// POUs/LinMot Config Function Blocks/LMcf_GetModUPIDList
FUNCTION_BLOCK LMcf_GetModUPIDList
VAR_INPUT
	Execute			:BOOL; 	(*Execute command*)
	adrFirstEntry	:POINTER TO tstLM_CfgUPIDListEntry; (*Points to the first entry of an array of UPIDListEntries (UPIDs and the according UPID values)*)
	NrOfEntries		:UINT; 	(*Number of parameters to be read. ATTENTION: Make sure the array at FirstEntry is big enough!!!!!*)
END_VAR
VAR_IN_OUT
	Axis			:tstLM_Axis; (*Axis reference*)
END_VAR
VAR_OUTPUT
	Done			:BOOL;	(*Command has been executed*)
	Busy			:BOOL;	(*Command running / FB Busy*)
	Error			:BOOL;	(*Error occured in FB*)
	ErrorID			:UINT;	(*Error ID:
							01h: Timeout (No Response from the drive)
							02h: ConfigChannel already busy
							05h: NrOfEntries must be greater than 0 (zero)! (UPID List)
							06h: Address of UPIDListEntry array is zero! Check adrFirstEntry input! (UPID List)
 							C0h: UPID Error 
 							C1h: Parameter Type Error
 							C2h: Range Error
 							C3h: Address Usage Error
 							C5h: Error: Command 21h
 							D0h: Odd Address
 							D1h: Size Error (Curve Service)
 							D4h: Curve already defined / Curve not present (Curve Service)
							>D4h: Contact LinMot Support
							*)
END_VAR
VAR
	uiState			:UINT;	(*internal -> *)
	i				:UINT;	(*internal -> *)
	pEntry			:POINTER TO tstLM_CfgUPIDListEntry; (*internal -> *)
	fStartTrig		:LM_R_TRIG;	(*internal -> *)
	fTimer			:TON;	(*internal -> *)
	tiT1			:TIME:=T#5000ms; (*internal -> timeout*)
END_VAR
(*Version history:
Date         	 | Version    	| Created under     		| Author          		| Remark 
------------------------------------------------------------------------------------------------------------------------------- 
2011-jul-12   	 | 1.0.0      	| V2.11.0 (Build 1016)		| fj  					| initial release 
*)

(*Check on errors*)
IF ((SHR(Axis.DrvToPlc.CfgStatusWord,8) = 16#C0)
	OR (SHR(Axis.DrvToPlc.CfgStatusWord,8) = 16#C1)
	OR (SHR(Axis.DrvToPlc.CfgStatusWord,8) = 16#C2)
	OR (SHR(Axis.DrvToPlc.CfgStatusWord,8) = 16#C3)
	OR (SHR(Axis.DrvToPlc.CfgStatusWord,8) = 16#C5)
	OR (SHR(Axis.DrvToPlc.CfgStatusWord,8) = 16#D0)
	OR (SHR(Axis.DrvToPlc.CfgStatusWord,8) = 16#D1)
	OR (SHR(Axis.DrvToPlc.CfgStatusWord,8) = 16#D4)
	OR (SHR(Axis.DrvToPlc.CfgStatusWord,8) > 16#D4))
	AND uiState > 1
	AND Busy THEN
	ErrorID := SHR(Axis.DrvToPlc.CfgStatusWord, 8);
	uiState := 90;
END_IF

(*Check start trigger*)
fStartTrig(CLK:=Execute);
IF fStartTrig.Q AND NOT Busy THEN
	IF Axis.ConfigChannelBusy THEN (*Check ConfigChannel busy*)
		ErrorID := 16#02; (*Error: ConfigChannel already busy*)
		uiState := 90; (*Error*)
	ELSIF NrOfEntries <= 0 THEN
		ErrorID := 16#05; (*Error: NrOfEntries must be greater than 0 (zero)! (UPID List)*)
		uiState := 90; (*Error*)
	ELSIF adrFirstEntry = 0 THEN
		ErrorID := 16#06; (*Address of UPIDListEntry array is zero! Check adrFirstEntry input! (UPID List)*)
		uiState := 90; (*Error*)
	ELSE
		Axis.ConfigChannelBusy := TRUE;
		Busy := TRUE;
		uiState := 1;
	END_IF
END_IF

(*State machine*)
CASE uiState OF
	(*Idle state*)
	0: 	;

(*=============================================================================
*  Get Modified UPID List
===============================================================================*)

	(*Prepare Config Module*)
	1: 	Axis.PlcToDrv.CfgControlWord := 16#000F;
		Axis.PlcToDrv.CfgIndexOut := 16#0000;
		Axis.PlcToDrv.CfgValueOut := 16#00000000;
		fTimer(IN:=TRUE,PT:=tiT1);

		pEntry := adrFirstEntry; (*Copy pointer*)
		i := 0; (*Reset i*)

		IF fTimer.Q THEN
			fTimer(IN:=FALSE);
			ErrorID := 16#01; (*fTimer error: No response from drive*)
			uiState := 90;
		END_IF

		IF Axis.DrvToPlc.CfgStatusWord = 16#000F THEN
			fTimer(IN:=FALSE);
			uiState := 2;
		END_IF

	 (*Start Getting Modified UPID List*)
	2:	Axis.PlcToDrv.CfgControlWord := 16#2201;
		fTimer(IN:=TRUE,PT:=tiT1);

		IF fTimer.Q THEN
			fTimer(IN:=FALSE);
			ErrorID := 16#01; (*fTimer error: No response from drive*)
			uiState := 90;
		END_IF

		IF Axis.DrvToPlc.CfgStatusWord = 16#0001 THEN
			fTimer(IN:=FALSE);
			uiState := 3;
		END_IF

	 (*Get Next Modified UPID List Item*)
	3:	Axis.PlcToDrv.CfgControlWord := 16#2302;
		fTimer(IN:=TRUE,PT:=tiT1);

		IF fTimer.Q THEN
			fTimer(IN:=FALSE);
			ErrorID := 16#01; (*fTimer error: No response from drive*)
			uiState := 90;
		END_IF

		IF Axis.DrvToPlc.CfgStatusWord = 16#C602 THEN (*End of UPID list reached*)
			fTimer(IN:=FALSE);
			pEntry^.UPID := Axis.DrvToPlc.CfgIndexIn; (*Read last UPID*)
			pEntry^.UPIDValue := Axis.DrvToPlc.CfgValueIn;
			i := i+1;
			uiState := 100;
		ELSIF Axis.DrvToPlc.CfgStatusWord = 16#0002 THEN (*UPID found*)
			fTimer(IN:=FALSE);
			pEntry^.UPID := Axis.DrvToPlc.CfgIndexIn;
			pEntry^.UPIDValue := Axis.DrvToPlc.CfgValueIn;
			pEntry := pEntry + (SIZEOF(adrFirstEntry^)); (*Increment pointer*)	
			i := i+1;
			IF i >= NrOfEntries THEN
				uiState := 100; (*Stop reading*)
			ELSE
				uiState := 4; (*Read next UPID*)
			END_IF
		END_IF

	(*Get Next Modified UPID List Item*)
	4:	Axis.PlcToDrv.CfgControlWord := 16#2303;
		fTimer(IN:=TRUE,PT:=tiT1);

		IF fTimer.Q THEN
			fTimer(IN:=FALSE);
			ErrorID := 16#01; (*fTimer error: No response from drive*)
			uiState := 90;
		END_IF

		IF Axis.DrvToPlc.CfgStatusWord = 16#C603 THEN (*End of UPID list reached*)
			fTimer(IN:=FALSE);
			pEntry^.UPID := Axis.DrvToPlc.CfgIndexIn; (*Read last UPID*)
			pEntry^.UPIDValue := Axis.DrvToPlc.CfgValueIn;
			i := i+1;
			uiState := 100;
		ELSIF Axis.DrvToPlc.CfgStatusWord = 16#0003 THEN (*UPID found*)
			fTimer(IN:=FALSE);
			pEntry^.UPID := Axis.DrvToPlc.CfgIndexIn;
			pEntry^.UPIDValue := Axis.DrvToPlc.CfgValueIn;
			pEntry := pEntry + (SIZEOF(adrFirstEntry^)); (*Increment pointer*)	
			i := i+1;
			IF i >= NrOfEntries THEN
				uiState := 100; (*Stop reading*)
			ELSE
				uiState := 3; (*Read next UPID*)
			END_IF
		END_IF

(*=============================================================================
*  Error State
===============================================================================*)    

	(*Error state I*)
	90:	IF Busy THEN
			Axis.ConfigChannelBusy := FALSE; (*Only reset ConfigChannelBusy if function block is Busy*)
			Axis.PlcToDrv.CfgControlWord := 16#0000; (*Reset Config Control*)
		END_IF

		Error := TRUE;
		Busy := FALSE;
		Done := FALSE;
		fTimer(IN:=FALSE);
		(*i := 0;*)

		uiState := 91;

	(*Error State II*)
	91:	IF NOT Execute THEN
			Error := FALSE;
			ErrorID := 0;
			uiState := 0;
		END_IF

(*=============================================================================
*  Command Done
===============================================================================*)    

	(*Command succesfully executed*)
	100:Done := TRUE;
		Busy := FALSE;
		fTimer(IN:=FALSE);
		(*i := 0;*)

		Axis.ConfigChannelBusy := FALSE;
		Axis.PlcToDrv.CfgControlWord := 16#0000; (*Reset Config Control*)

		uiState := 101;

	(*Wait Not Execute*)
	101:IF NOT Execute THEN
			Done := FALSE;
			uiState := 0;
		END_IF

END_CASE

END_FUNCTION_BLOCK

// POUs/LinMot Config Function Blocks/LMcf_ParaAccess
FUNCTION_BLOCK LMcf_ParaAccess
VAR_INPUT
	Execute			:BOOL;	(*Execute command*)
	Mode			:UINT;	(*Mode 0: Read ROM Value of Parameter by UPID [Inputs used: UPIDIn]
 							Mode 1: Read RAM Value of Parameter by UPID [Inputs used: UPIDIn]
 							Mode 2: Write ROM Value of Parameter by UPID [Inputs used: UPIDIn, ValueIn]
 							Mode 3: Write RAM Value of Parameter by UPID [Inputs used: UPIDIn, ValueIn]
 							Mode 4: Write RAM and ROM Value of Parameter by UPID [Inputs used: UPIDIn, ValueIn]
 							Mode 5: Get minimal Value of Parameter by UPID [Inputs used: UPIDIn]
 							Mode 6: Get maximal Value of Parameter by UPID [Inputs used: UPIDIn]
 							Mode 7: Get default Value of Parameter by UPID [Inputs used: UPIDIn]
							*)
	UPIDIn			:UINT;	(*UPID to access*)
	ValueIn			:DINT;	(*UPID value to be written*)
END_VAR
VAR_IN_OUT
	Axis			:tstLM_Axis; (*Axis reference*)
END_VAR
VAR_OUTPUT
	Done			:BOOL;	(*Command has been executed*)
	Busy			:BOOL;	(*Command running / FB Busy*)
	ValueOut		:DINT;	(*UPID value from drive*)
	Error			:BOOL;	(*Error occured in FB*)
	ErrorID			:UINT;	(*Error ID:
							01h: Timeout (No Response from the drive)
							02h: ConfigChannel already busy
							03h: Invalid Mode selected
 							C0h: UPID Error 
 							C1h: Parameter Type Error
 							C2h: Range Error
 							C3h: Address Usage Error
 							C5h: Error: Command 21h
 							D0h: Odd Address
 							D1h: Size Error (Curve Service)
 							D4h: Curve already defined / Curve not present (Curve Service)
							>D4h: Contact LinMot Support
							*)
END_VAR
VAR
	uiState			:UINT;	(*internal -> *)
	uiStartState	:UINT;	(*internal -> *)
	fStartTrig		:LM_R_TRIG;	(*internal -> *)
	fTimer			:TON;	(*internal -> *)
	tiT1			:TIME:=T#5000MS; (*internal -> timeout*)
END_VAR
(*Version history:
Date         	 | Version    	| Created under     		| Author          		| Remark 
------------------------------------------------------------------------------------------------------------------------------- 
2011-jul-12   	 | 1.0.0      		| V2.11.0 (Build 1016)	| fj  				| initial release 
*)

(*Check on errors*)
IF ((SHR(Axis.DrvToPlc.CfgStatusWord,8) = 16#C0)
	OR (SHR(Axis.DrvToPlc.CfgStatusWord,8) = 16#C1)
	OR (SHR(Axis.DrvToPlc.CfgStatusWord,8) = 16#C2)
	OR (SHR(Axis.DrvToPlc.CfgStatusWord,8) = 16#C3)
	OR (SHR(Axis.DrvToPlc.CfgStatusWord,8) = 16#C5)
	OR (SHR(Axis.DrvToPlc.CfgStatusWord,8) = 16#D0)
	OR (SHR(Axis.DrvToPlc.CfgStatusWord,8) = 16#D1)
	OR (SHR(Axis.DrvToPlc.CfgStatusWord,8) = 16#D4)
	OR (SHR(Axis.DrvToPlc.CfgStatusWord,8) > 16#D4))
	AND uiState > 1
	AND Busy THEN
	ErrorID := SHR(Axis.DrvToPlc.CfgStatusWord, 8);
	uiState := 90;
END_IF

(*Mode selection and edge detection*)
fStartTrig(CLK:=Execute);
IF fStartTrig.Q AND NOT Busy THEN
	CASE Mode OF
		(*Read ROM Value of Parameter by UPID*)
		0: 	uiStartState := 2;
			uiState := 1;
		(*Read RAM Value of Parameter by UPID*)
		1: 	uiStartState := 10;
			uiState := 1;
		(*Write ROM Value of Parameter by UPID*)
		2: 	uiStartState := 20;
			uiState := 1;
		(*Write RAM Value of Parameter by UPID*)
		3: 	uiStartState := 30;
			uiState := 1;
		(*Write RAM and ROM Value of Parameter by UPID*)
		4: 	uiStartState := 40;
			uiState := 1;
		(*Get minimal Value of Parameter by UPID*)
		5: 	uiStartState := 50;
			uiState := 1;
		(*Get maximal Value of Parameter by UPID*)
		6: 	uiStartState := 60;
			uiState := 1;
		(*Get default Value of Parameter by UPID*)
		7: 	uiStartState := 70;
			uiState := 1;
		ELSE ;
	END_CASE

	IF Axis.ConfigChannelBusy THEN (*Check ConfigChannel busy*)
		ErrorID := 16#02; (*Error: ConfigChannel already busy*)
		uiState := 90; (*Error*)
	ELSIF Mode > 7 THEN
		ErrorID := 16#03; (*Error: Invalid Mode selected*)
		uiState := 90; (*Error*)
	ELSE
		Axis.ConfigChannelBusy := TRUE;
		Busy := TRUE;
	END_IF
END_IF

(*State machine*)
CASE uiState OF
	(*Idle state*)
	0: 	;

	(*Prepare Config Module*)
	1: 	Axis.PlcToDrv.CfgControlWord := 16#000F;
		Axis.PlcToDrv.CfgIndexOut := 16#0000;
		Axis.PlcToDrv.CfgValueOut := 16#00000000;
		fTimer(IN:=TRUE,PT:=tiT1);

		IF fTimer.Q THEN
			fTimer(IN:=FALSE);
			ErrorID := 16#01; (*fTimer error: No response from drive*)
			uiState := 90;
		END_IF

		IF Axis.DrvToPlc.CfgStatusWord = 16#000F THEN
			fTimer(IN:=FALSE);
			uiState := uiStartState;
		END_IF

(*=============================================================================
*  Mode 0: 
*  Read ROM Value of Parameter by UPID
===============================================================================*)    

	 (*Read ROM Value of Parameter by UPID*)
	2:	Axis.PlcToDrv.CfgControlWord := 16#1001;
		Axis.PlcToDrv.CfgIndexOut := UPIDIn;
		fTimer(IN:=TRUE,PT:=tiT1);

		IF fTimer.Q THEN
			fTimer(IN:=FALSE);
			ErrorID := 16#01; (*fTimer error: No response from drive*)
			uiState := 90;
		END_IF

		IF Axis.DrvToPlc.CfgStatusWord = 16#0001 THEN
			ValueOut := UDINT_TO_DINT(Axis.DrvToPlc.CfgValueIn);
			fTimer(IN:=FALSE);
			uiState := 100;
		END_IF

(*=============================================================================
*  Mode 1: 
*  Read RAM Value of Parameter by UPID
===============================================================================*)    

	 (*Read RAM Value of Parameter by UPID*)
	10:	Axis.PlcToDrv.CfgControlWord := 16#1101;
		Axis.PlcToDrv.CfgIndexOut := UPIDIn;
		fTimer(IN:=TRUE,PT:=tiT1);

		IF fTimer.Q THEN
			fTimer(IN:=FALSE);
			ErrorID := 16#01; (*fTimer error: No response from drive*)
			uiState := 90;
		END_IF

		IF Axis.DrvToPlc.CfgStatusWord = 16#0001THEN
			fTimer(IN:=FALSE);
			ValueOut := UDINT_TO_DINT(Axis.DrvToPlc.CfgValueIn);
			uiState := 100;
		END_IF

(*=============================================================================
*  Mode 2: 
*  Write ROM Value of Parameter by UPID
===============================================================================*)    

	 (*Write ROM Value of Parameter by UPID*)
	20:	Axis.PlcToDrv.CfgControlWord := 16#1201;
		Axis.PlcToDrv.CfgIndexOut := UPIDIn;
		Axis.PlcToDrv.CfgValueOut := DINT_TO_UDINT(ValueIn);
		fTimer(IN:=TRUE,PT:=tiT1);

		IF fTimer.Q THEN
			fTimer(IN:=FALSE);
			ErrorID := 16#01; (*fTimer error: No response from drive*)
			uiState := 90;
		END_IF

		IF Axis.DrvToPlc.CfgStatusWord = 16#0001 THEN
			fTimer(IN:=FALSE);
			ValueOut := UDINT_TO_DINT(Axis.DrvToPlc.CfgValueIn);
			uiState := 100;
		END_IF

(*=============================================================================
*  Mode 3: 
*  Write RAM Value of Parameter by UPID
===============================================================================*)    

	 (*Write RAM Value of Parameter by UPID*)
	30:	Axis.PlcToDrv.CfgControlWord := 16#1301;
		Axis.PlcToDrv.CfgIndexOut := UPIDIn;
		Axis.PlcToDrv.CfgValueOut := DINT_TO_UDINT(ValueIn);
		fTimer(IN:=TRUE,PT:=tiT1);

		IF fTimer.Q THEN
			fTimer(IN:=FALSE);
			ErrorID := 16#01; (*fTimer error: No response from drive*)
			uiState := 90;
		END_IF

		IF Axis.DrvToPlc.CfgStatusWord = 16#0001 THEN
			fTimer(IN:=FALSE);
			ValueOut := UDINT_TO_DINT(Axis.DrvToPlc.CfgValueIn);
			uiState := 100;
		END_IF

(*=============================================================================
*  Mode 4: 
*  Write RAM and ROM Value of Parameter by UPID
===============================================================================*)    

	 (*Write RAM and ROM Value of Parameter by UPID*)
	40:	Axis.PlcToDrv.CfgControlWord := 16#1401;
		Axis.PlcToDrv.CfgIndexOut :=  UPIDIn;
		Axis.PlcToDrv.CfgValueOut := DINT_TO_UDINT(ValueIn);
		fTimer(IN:=TRUE,PT:=tiT1);

		IF fTimer.Q THEN
			fTimer(IN:=FALSE);
			ErrorID := 16#01; (*fTimer error: No response from drive*)
			uiState := 90;
		END_IF

		IF Axis.DrvToPlc.CfgStatusWord = 16#0001 THEN
			fTimer(IN:=FALSE);
			ValueOut := UDINT_TO_DINT(Axis.DrvToPlc.CfgValueIn);
			uiState := 100;
		END_IF

(*=============================================================================
*  Mode 5: 
* Get minimal Value of Parameter by UPID
===============================================================================*)    

	(*Get minimal Value of Parameter by UPID*)
	50:	Axis.PlcToDrv.CfgControlWord := 16#1501;
		Axis.PlcToDrv.CfgIndexOut := UPIDIn;
		fTimer(IN:=TRUE,PT:=tiT1);

		IF fTimer.Q THEN
			fTimer(IN:=FALSE);
			ErrorID := 16#01; (*fTimer error: No response from drive*)
			uiState := 90;
		END_IF

		IF Axis.DrvToPlc.CfgStatusWord = 16#0001 THEN
			fTimer(IN:=FALSE);
			ValueOut := UDINT_TO_DINT(Axis.DrvToPlc.CfgValueIn);
			uiState := 100;
		END_IF

(*=============================================================================
*  Mode 6: 
* Get maximal Value of Parameter by UPID
===============================================================================*)    

	 (*Get maximal Value of Parameter by UPID*)
	60:	Axis.PlcToDrv.CfgControlWord := 16#1601;
		Axis.PlcToDrv.CfgIndexOut := UPIDIn;
		fTimer(IN:=TRUE,PT:=tiT1);

		IF fTimer.Q THEN
			fTimer(IN:=FALSE);
			ErrorID := 16#01; (*fTimer error: No response from drive*)
			uiState := 90;
		END_IF

		IF Axis.DrvToPlc.CfgStatusWord = 16#0001 THEN
			fTimer(IN:=FALSE);
			ValueOut := UDINT_TO_DINT(Axis.DrvToPlc.CfgValueIn);
			uiState := 100;
		END_IF

(*=============================================================================
*  Mode 7: 
* Get default Value of Parameter by UPID
===============================================================================*)    

	 (*Get default Value of Parameter by UPID*)
	70:	Axis.PlcToDrv.CfgControlWord := 16#1701;
		Axis.PlcToDrv.CfgIndexOut := UPIDIn;
		fTimer(IN:=TRUE,PT:=tiT1);

		IF fTimer.Q THEN
			fTimer(IN:=FALSE);
			ErrorID := 16#01; (*fTimer error: No response from drive*)
			uiState := 90;
		END_IF

		IF Axis.DrvToPlc.CfgStatusWord = 16#0001 THEN
			fTimer(IN:=FALSE);
			ValueOut := UDINT_TO_DINT(Axis.DrvToPlc.CfgValueIn);
			uiState := 100;
		END_IF

(*=============================================================================
*  Error State
===============================================================================*)    

	(*Error state I*)
	90:	IF Busy THEN
			Axis.ConfigChannelBusy := FALSE; (*Only reset ConfigChannelBusy if function block is Busy*)
			Axis.PlcToDrv.CfgControlWord := 16#0000; (*Reset Config Control*)
		END_IF

		Error := TRUE;
		Busy := FALSE;
		Done := FALSE;
		ValueOut := 0;
		fTimer(IN:=FALSE);

		uiState := 91;

	(*Error State II*)
	91:	IF NOT Execute THEN
			Error := FALSE;
			ErrorID := 0;
			uiState := 0;
		END_IF

(*=============================================================================
*  Command Done
===============================================================================*)    

	(*Command succesfully executed*)
	100:Done := TRUE;
		Busy := FALSE;
		fTimer(IN:=FALSE);

		Axis.ConfigChannelBusy := FALSE;
		Axis.PlcToDrv.CfgControlWord := 16#0000; (*Reset Config Control*)

		uiState := 101;

	(*Wait Not Execute*)
	101:IF NOT Execute THEN
			Done := FALSE;
			ValueOut := 0;
			uiState := 0;
		END_IF

END_CASE

END_FUNCTION_BLOCK

// POUs/LinMot Config Function Blocks/LMcf_StopStartDefault
FUNCTION_BLOCK LMcf_StopStartDefault
VAR_INPUT
	Execute			:BOOL;	(*Execute command*)
	Mode			:UINT;	(*Mode 0: Restart drive
 							Mode 1: Set parameter ROM values to default (OS SW)
 							Mode 2: Set parameter ROM values to default (MC SW)
 							Mode 3: Set parameter ROM values to default (Interface SW)
							Mode 4: Set parameter ROM values to default (Application SW)_ __					
							Mode 5: Stop MC and Application Software (for Flash Access)
 							Mode 6: Start MC and Application Software 
							*)
END_VAR
VAR_IN_OUT
	Axis			:tstLM_Axis; (*Axis reference*)
END_VAR
VAR_OUTPUT
	Done			:BOOL;	(*Command has been executed*)
	Busy			:BOOL;	(*Command running / FB Busy*)
	Error			:BOOL;	(*Error occured in FB*)
	ErrorID			:UINT;	(*Error ID:
							01h: Timeout (No Response from the drive)
							02h: ConfigChannel already busy
							03h: Invalid Mode selected
 							C0h: UPID Error 
 							C1h: Parameter Type Error
 							C2h: Range Error
 							C3h: Address Usage Error
 							C5h: Error: Command 21h
 							D0h: Odd Address
 							D1h: Size Error (Curve Service)
 							D4h: Curve already defined / Curve not present (Curve Service)
							>D4h: Contact LinMot Support
							*)
END_VAR
VAR
	uiState			:UINT;	(*internal -> *)
	uiStartState	:UINT;	(*internal -> *)
	fStartTrig		:LM_R_TRIG;	(*internal -> *)
	fTimer			:TON;	(*internal -> *)
	tiT1			:TIME:=T#60000MS; (*internal -> timeout*)
END_VAR
(*Version history:
Date         	 | Version    	| Created under     		| Author          		| Remark 
------------------------------------------------------------------------------------------------------------------------------- 
2011-jul-12   	 | 1.0.0      		| V2.11.0 (Build 1016)	| fj  				| initial release 
*)

(*Check on errors*)
IF ((SHR(Axis.DrvToPlc.CfgStatusWord,8) = 16#C0)
	OR (SHR(Axis.DrvToPlc.CfgStatusWord,8) = 16#C1)
	OR (SHR(Axis.DrvToPlc.CfgStatusWord,8) = 16#C2)
	OR (SHR(Axis.DrvToPlc.CfgStatusWord,8) = 16#C3)
	OR (SHR(Axis.DrvToPlc.CfgStatusWord,8) = 16#C5)
	OR (SHR(Axis.DrvToPlc.CfgStatusWord,8) = 16#D0)
	OR (SHR(Axis.DrvToPlc.CfgStatusWord,8) = 16#D1)
	OR (SHR(Axis.DrvToPlc.CfgStatusWord,8) = 16#D4)
	OR (SHR(Axis.DrvToPlc.CfgStatusWord,8) > 16#D4))
	AND uiState > 1
	AND Busy THEN
	ErrorID := SHR(Axis.DrvToPlc.CfgStatusWord, 8);
	uiState := 90;
END_IF

(*Mode selection and edge detection*)
fStartTrig(CLK:=Execute);
IF fStartTrig.Q AND NOT Busy THEN
	CASE Mode OF
		(*Restart drive*)
		0: 	uiStartState := 2;
			uiState := 1;
		(*Set parameter ROM values to default (OS SW)*)
		1: 	uiStartState := 10;
			uiState := 1;
		(*Set parameter ROM values to default (MC SW)*)
		2: 	uiStartState := 20;
			uiState := 1;
		(*Set parameter ROM values to default (Interface SW)*)
		3: 	uiStartState := 30;
			uiState := 1;
		(*Set parameter ROM values to default (Application SW)*)
		4: 	uiStartState := 40;
			uiState := 1;
		(*Stop MC and Application Software (for Flash Access)*)
		5: 	uiStartState := 50;
			uiState := 1;
		(*Start MC and Application Software*)
		6: 	uiStartState := 60;
			uiState := 1;
		ELSE ;
	END_CASE

	IF Axis.ConfigChannelBusy THEN (*Check ConfigChannel busy*)
		ErrorID := 16#02; (*Error: ConfigChannel already busy*)
		uiState := 90; (*Error*)
	ELSIF Mode > 6 THEN
		ErrorID := 16#03; (*Error: Invalid Mode selected*)
		uiState := 90; (*Error*)
	ELSE
		Axis.ConfigChannelBusy := TRUE;
		Busy := TRUE;
	END_IF
END_IF

(*State machine*)
CASE uiState OF
	(*Idle state*)
	0: 	;

	(*Prepare Config Module*)
	1: 	Axis.PlcToDrv.CfgControlWord := 16#000F;
		Axis.PlcToDrv.CfgIndexOut := 16#0000;
		Axis.PlcToDrv.CfgValueOut := 16#00000000;
		fTimer(IN:=TRUE,PT:=tiT1);

		IF fTimer.Q THEN
			fTimer(IN:=FALSE);
			ErrorID := 16#01; (*fTimer error: No response from drive*)
			uiState := 90;
		END_IF

		IF Axis.DrvToPlc.CfgStatusWord = 16#000F THEN
			fTimer(IN:=FALSE);
			uiState := uiStartState;
		END_IF

(*=============================================================================
*  Mode 0: 
*  Restart drive
===============================================================================*)    

	 (*Restart drive*)
	2:	Axis.PlcToDrv.CfgControlWord := 16#3000;
		fTimer(IN:=TRUE,PT:=tiT1);

		IF fTimer.Q THEN
			fTimer(IN:=FALSE);
			ErrorID := 16#01; (*fTimer error: No response from drive*)
			uiState := 90;
		END_IF

		IF Axis.DrvToPlc.CfgStatusWord = 16#0000 THEN
			fTimer(IN:=FALSE);
			uiState := 3;
		END_IF

	 (*Restart drive II*)
	3:	Axis.PlcToDrv.CfgControlWord := 16#0001; (*Poll drive to check if reboot has been completed*)
		fTimer(IN:=TRUE,PT:=tiT1);

		IF fTimer.Q THEN
			fTimer(IN:=FALSE);
			ErrorID := 16#01; (*fTimer error: No response from drive*)
			uiState := 90;
		END_IF

		IF Axis.DrvToPlc.CfgStatusWord = 16#0001 THEN
			fTimer(IN:=FALSE);
			uiState := 100;
		END_IF

(*=============================================================================
*  Mode 1: 
*  Set parameter ROM values to default (OS SW)
===============================================================================*)    

	 (*Set parameter ROM values to default (OS SW)*)
	10:	Axis.PlcToDrv.CfgControlWord := 16#3100;
		fTimer(IN:=TRUE,PT:=tiT1);

		IF fTimer.Q THEN
			fTimer(IN:=FALSE);
			ErrorID := 16#01; (*fTimer error: No response from drive*)
			uiState := 90;
		END_IF

		IF Axis.DrvToPlc.CfgStatusWord = 16#0000 THEN
			fTimer(IN:=FALSE);
			uiState := 100;
		END_IF

(*=============================================================================
*  Mode 2: 
*  Set parameter ROM values to default (MC SW)
===============================================================================*)    

	 (*Set parameter ROM values to default (MC SW)*)
	20:	Axis.PlcToDrv.CfgControlWord := 16#3200;
		fTimer(IN:=TRUE,PT:=tiT1);

		IF fTimer.Q THEN
			fTimer(IN:=FALSE);
			ErrorID := 16#01; (*fTimer error: No response from drive*)
			uiState := 90;
		END_IF

		IF Axis.DrvToPlc.CfgStatusWord = 16#0000 THEN
			fTimer(IN:=FALSE);
			uiState := 100;
		END_IF

(*=============================================================================
*  Mode 3: 
*  Set parameter ROM values to default (Interface SW)
===============================================================================*)    

	 (*Set parameter ROM values to default (Interface SW)*)
	30:	Axis.PlcToDrv.CfgControlWord := 16#3300;
		fTimer(IN:=TRUE,PT:=tiT1);

		IF fTimer.Q THEN
			fTimer(IN:=FALSE);
			ErrorID := 16#01; (*fTimer error: No response from drive*)
			uiState := 90;
		END_IF

		IF Axis.DrvToPlc.CfgStatusWord = 16#0000 THEN
			fTimer(IN:=FALSE);
			uiState := 100;
		END_IF

(*=============================================================================
*  Mode 4: 
*  Set parameter ROM values to default (Application SW)
===============================================================================*)    

	(*Set parameter ROM values to default (Application SW)*)
	40:	Axis.PlcToDrv.CfgControlWord := 16#3400;
		fTimer(IN:=TRUE,PT:=tiT1);

		IF fTimer.Q THEN
			fTimer(IN:=FALSE);
			ErrorID := 16#01; (*fTimer error: No response from drive*)
			uiState := 90;
		END_IF

		IF Axis.DrvToPlc.CfgStatusWord = 16#0000 THEN
			fTimer(IN:=FALSE);
			uiState := 100;
		END_IF

(*=============================================================================
*  Mode 5: 
* Stop MC and Application Software (for Flash Access)
===============================================================================*)    

	(*Stop MC and Application Software (for Flash Access)*)
	50:	Axis.PlcToDrv.CfgControlWord := 16#3500;
		fTimer(IN:=TRUE,PT:=tiT1);

		IF fTimer.Q THEN
			fTimer(IN:=FALSE);
			ErrorID := 16#01; (*fTimer error: No response from drive*)
			uiState := 90;
		END_IF

		IF Axis.DrvToPlc.CfgStatusWord = 16#0000 THEN
			fTimer(IN:=FALSE);
			uiState := 100;
		END_IF

(*=============================================================================
*  Mode 6: 
* Start MC and Application Software
===============================================================================*)    

	(*Start MC and Application Software*)
	60:	Axis.PlcToDrv.CfgControlWord := 16#3600;
		fTimer(IN:=TRUE,PT:=tiT1);

		IF fTimer.Q THEN
			fTimer(IN:=FALSE);
			ErrorID := 16#01; (*fTimer error: No response from drive*)
			uiState := 90;
		END_IF

		IF Axis.DrvToPlc.CfgStatusWord = 16#0000 THEN
			fTimer(IN:=FALSE);
			uiState := 100;
		END_IF

(*=============================================================================
*  Error State
===============================================================================*)    

	(*Error State I*)
	90:	IF Busy THEN
			Axis.ConfigChannelBusy := FALSE; (*Only reset ConfigChannelBusy if function block is Busy*)
			Axis.PlcToDrv.CfgControlWord := 16#0000; (*Reset Config Control*)
		END_IF

		Error := TRUE;
		Busy := FALSE;
		Done := FALSE;
		fTimer(IN:=FALSE);

		uiState := 91;

	(*Error State II*)
	91:	IF NOT Execute THEN
			Error := FALSE;
			ErrorID := 0;
			uiState := 0;
		END_IF

(*=============================================================================
*  Command Done
===============================================================================*)    

	(*Command succesfully executed*)
	100:Done := TRUE;
		Busy := FALSE;
		fTimer(IN:=FALSE);

		Axis.ConfigChannelBusy := FALSE;
		Axis.PlcToDrv.CfgControlWord := 16#0000; (*Reset Config Control*)

		uiState := 101;

	(*Wait Not Execute*)
	101:IF NOT Execute THEN
			Done := FALSE;
			uiState := 0;
		END_IF

END_CASE

END_FUNCTION_BLOCK

// POUs/LinMot Config Function Blocks/LMcf_WriteUPIDList
FUNCTION_BLOCK LMcf_WriteUPIDList
VAR_INPUT
	Execute			:BOOL; 	(*Execute command*)
	adrFirstEntry	:POINTER TO tstLM_CfgUPIDListEntry; (*Points to the first entry of an array of UPIDListEntries (UPIDs and the according UPID values)*)
	NrOfEntries		:UINT; 	(*Number of parameters to be read. ATTENTION: Make sure the array at FirstEntry is big enough!!!!!*)
END_VAR
VAR_IN_OUT
	Axis			:tstLM_Axis; (*Axis reference*)
END_VAR
VAR_OUTPUT
	Done			:BOOL;	(*Command has been executed*)
	Busy			:BOOL;	(*Command running / FB Busy*)
	Error			:BOOL;	(*Error occured in FB*)
	ErrorID			:UINT;	(*Error ID:
							01h: Timeout (No Response from the drive)
							02h: ConfigChannel already busy
							05h: NrOfEntries must be greater than 0 (zero)! (UPID List)
							06h: Pointer to UPIDListEntry array is zero! Check adrFirstEntry input! (UPID List)
 							C0h: UPID Error 
 							C1h: Parameter Type Error
 							C2h: Range Error
 							C3h: Address Usage Error
 							C5h: Error: Command 21h
 							D0h: Odd Address
 							D1h: Size Error (Curve Service)
 							D4h: Curve already defined / Curve not present (Curve Service)
							>D4h: Contact LinMot Support
							*)
END_VAR
VAR
	uiState			:UINT;	(*internal -> *)
	i				:UINT;	(*internal -> *)
	pEntry			:POINTER TO tstLM_CfgUPIDListEntry; (*internal -> *)
	fStartTrig		:LM_R_TRIG;	(*internal -> *)
	fTimer			:TON;	(*internal -> *)
	tiT1			:TIME:=T#5000MS; (*internal -> timeout*)
END_VAR
(*Version history:
Date         	 | Version    	| Created under     		| Author          		| Remark 
------------------------------------------------------------------------------------------------------------------------------- 
2011-jul-12   	 | 1.0.0      		| V2.11.0 (Build 1016)	| fj  				| initial release 
*)

(*Check on errors*)
IF ((SHR(Axis.DrvToPlc.CfgStatusWord,8) = 16#C0)
	OR (SHR(Axis.DrvToPlc.CfgStatusWord,8) = 16#C1)
	OR (SHR(Axis.DrvToPlc.CfgStatusWord,8) = 16#C2)
	OR (SHR(Axis.DrvToPlc.CfgStatusWord,8) = 16#C3)
	OR (SHR(Axis.DrvToPlc.CfgStatusWord,8) = 16#C5)
	OR (SHR(Axis.DrvToPlc.CfgStatusWord,8) = 16#D0)
	OR (SHR(Axis.DrvToPlc.CfgStatusWord,8) = 16#D1)
	OR (SHR(Axis.DrvToPlc.CfgStatusWord,8) = 16#D4)
	OR (SHR(Axis.DrvToPlc.CfgStatusWord,8) > 16#D4))
	AND uiState > 1
	AND Busy THEN
	ErrorID := SHR(Axis.DrvToPlc.CfgStatusWord, 8);
	uiState := 90;
END_IF

(*Check start trigger*)
fStartTrig(CLK:=Execute);
IF fStartTrig.Q AND NOT Busy THEN
	IF Axis.ConfigChannelBusy THEN (*Check ConfigChannel busy*)
		ErrorID := 16#02; (*Error: ConfigChannel already busy*)
		uiState := 90; (*Error*)
	ELSIF NrOfEntries <= 0 THEN
		ErrorID := 16#05; (*Error: NrOfEntries must be greater than 0 (zero)! (UPID List)*)
		uiState := 90; (*Error*)
	ELSIF adrFirstEntry = 0 THEN
		ErrorID := 16#06; (*Error: Pointer to UPIDListEntry array is zero! Check adrFirstEntry input! (UPID List)*)
		uiState := 90; (*Error*)
	ELSE
		Axis.ConfigChannelBusy := TRUE;
		Busy := TRUE;
		uiState := 1;
	END_IF
END_IF

(*State machine*)
CASE uiState OF
	(*Idle state*)
	0: 	;

(*=============================================================================
*  Write UPID Array
===============================================================================*)

	(*Prepare Config Module*)
	1: 	Axis.PlcToDrv.CfgControlWord := 16#000F;
		Axis.PlcToDrv.CfgIndexOut := 16#0000;
		Axis.PlcToDrv.CfgValueOut := 16#00000000;
		fTimer(IN:=TRUE,PT:=tiT1);
		i := 0;
		pEntry := adrFirstEntry;

		IF fTimer.Q THEN
			fTimer(IN:=FALSE);
			ErrorID := 16#01; (*fTimer error: No response from drive*)
			uiState := 90;
		END_IF

		IF Axis.DrvToPlc.CfgStatusWord = 16#000F THEN
			fTimer(IN:=FALSE);
			uiState := 2;
		END_IF

	 (*Write UPID Value to ROM*)
	2:	IF Axis.DrvToPlc.CfgStatusWord = 16#0001 THEN (*UPID written*)
			 (*Prepare writing next UPID*)
			fTimer(IN:=FALSE);
			i := i+1;
			IF i >= NrOfEntries THEN (*All UPIDs written*)
				uiState := 100;
			ELSE	
				pEntry := pEntry + (SIZEOF(adrFirstEntry^)); (*Increment pointer*)			
				IF pEntry^.UPID = 0 THEN (*Check next UPID valid*)
					uiState := 100; (*Next UPID is zero -> Abort writing*)
				ELSE
					uiState := 3;
				END_IF
			END_IF
		END_IF

		IF uiState <> 100 THEN
			Axis.PlcToDrv.CfgControlWord := 16#1201;
			Axis.PlcToDrv.CfgIndexOut := pEntry^.UPID;
			Axis.PlcToDrv.CfgValueOut := pEntry^.UPIDValue;
			fTimer(IN:=TRUE,PT:=tiT1);
		END_IF

		IF fTimer.Q THEN
			fTimer(IN:=FALSE);
			ErrorID := 16#01; (*fTimer error: No response from drive*)
			uiState := 90;
		END_IF

	(*Write UPID Value to ROM*)
	3:	IF Axis.DrvToPlc.CfgStatusWord = 16#0002 THEN (*UPID written*)
			 (*Prepare writing next UPID*)
			fTimer(IN:=FALSE);
			i := i+1;
			IF i >= NrOfEntries THEN (*All UPIDs written*)
				uiState := 100;
			ELSE
				pEntry := pEntry + (SIZEOF(adrFirstEntry^)); (*Increment pointer*)	
				IF pEntry^.UPID = 0 THEN (*Check next UPID valid*)
					uiState := 100; (*Next UPID is zero -> Abort writing*)
				ELSE
					uiState := 2;
				END_IF
			END_IF
		END_IF

		IF uiState <> 100 THEN
			Axis.PlcToDrv.CfgControlWord := 16#1202;
			Axis.PlcToDrv.CfgIndexOut := pEntry^.UPID;
			Axis.PlcToDrv.CfgValueOut := pEntry^.UPIDValue;
			fTimer(IN:=TRUE,PT:=tiT1);
		END_IF

		IF fTimer.Q THEN
			fTimer(IN:=FALSE);
			ErrorID := 16#01; (*fTimer error: No response from drive*)
			uiState := 90;
		END_IF

(*=============================================================================
*  Error State
===============================================================================*)    

	(*Error State I*)
	90:	IF Busy THEN
			Axis.ConfigChannelBusy := FALSE; (*Only reset ConfigChannelBusy if function block is Busy*)
			Axis.PlcToDrv.CfgControlWord := 16#0000; (*Reset Config Control*)
		END_IF

		Error := TRUE;
		Busy := FALSE;
		Done := FALSE;
		fTimer(IN:=FALSE);
		(*i := 0;*)

		uiState := 91;

	(*Error State II*)
	91:	IF NOT Execute THEN
			Error := FALSE;
			ErrorID := 0;
			uiState := 0;
		END_IF

(*=============================================================================
*  Command Done
===============================================================================*)    

	(*Command succesfully executed*)
	100:Done := TRUE;
		Busy := FALSE;
		fTimer(IN:=FALSE);
		(*i := 0;*)

		Axis.ConfigChannelBusy := FALSE;
		Axis.PlcToDrv.CfgControlWord := 16#0000; (*Reset Config Control*)

		uiState := 101;

	(*Wait Not Execute*)
	101:IF NOT Execute THEN
			Done := FALSE;
			uiState := 0;
		END_IF

END_CASE

END_FUNCTION_BLOCK

// POUs/LinMot Force Control Function Blocks/Unofficial_Unsupported/LMfc_ChangeTargetForceCont
FUNCTION_BLOCK LMfc_ChangeTargetForceCont
VAR_INPUT
	Enable 			:BOOL;	(*Enable streaming*)
	TargetForce		:REAL;	(*Target force*)
END_VAR
VAR_IN_OUT
	Axis 			:tstLM_Axis; (*Axis reference*)
END_VAR
VAR_OUTPUT
	Streaming		:BOOL;	(*Streaming / FB Busy*)
	Error 			:BOOL;	(*Error detected*)
	ErrorID			:UINT;	(*Error ID:
							01h: Axis not ready
 							02h: Axis already has command running
 							03h: Axis has error
 							04h: Command interrupted
 							05h: Command aborted
							06h: Invalid input(s)
							*)
END_VAR
VAR
	uiCState		:UINT;	(*internal -> *)
	uiFbState 		:UINT;	(*internal -> *)
	rTrig			:LM_R_TRIG;	(*internal -> *)
	udiTmpDWord 	:UDINT;	(*internal -> *)
	bTemp 			:BOOL;	(*internal -> *)

 	uiCmdHeader 	:UINT := 16#3820;	(*CommandHeader (382xh) of the "Force Ctrl Change Target Force (382xh)" motion command*)
END_VAR
(*Version history:
Date         	 | Version    		| Created under     	| Author          	| Remark 
------------------------------------------------------------------------------------------------------------------------------- 
2011-sep-13   	 | 1.0.0      		| V2.11.0 (Build 1016)	| fj  				| initial release
2011-dec-01   	 | 1.0.2      		| V2.11.0 (Build 1016)	| fj  				| code optimisation
2012-apr-25   	 | 1.1.0     		| V2.11.0 (Build 1016)	| fj  				| added input parameters check
*)

(*Variablen ][ variables*)
	uiCState := SHR(Axis.DrvToPlc.StateVar, 8);

(*Flankenerkennung am Enable Eingang*)
(*Edge detection on Enable input*)
rTrig(CLK:=Enable);
IF rTrig.Q AND uiCState = 16#08 AND NOT Axis.CommandRunning THEN (*Start command*)
	Axis.CommandRunning := TRUE;
	uiFbState := 1;
ELSIF rTrig.Q AND uiCState <> 16#08 THEN (*Axis not ready*)
	uiFbState := 50; (*Error state*)
	Error := TRUE;
	ErrorID := 16#01; (*Axis not ready*)
ELSIF rTrig.Q AND Axis.CommandRunning THEN (*Axis already has a command running*)
	uiFbState := 50; (*Error state*)
	Error := TRUE;
	ErrorID := 16#02; (*Axis already has a command running*)
END_IF

IF Streaming AND uiCState = 16#04 THEN
	Axis.CommandRunning := FALSE;
	uiFbState := 50;
	Error := TRUE;
	ErrorID := 16#03; (*Axis has error*)
END_IF

IF Streaming AND uiCState <> 16#08 THEN
	Axis.CommandRunning := FALSE;
	uiFbState := 50; (*Error state*)
	Error := TRUE;
	ErrorID := 16#04; (*Command interupted*)
ELSIF Streaming AND Axis.CommandAborted THEN
	uiFbState := 50; (*Error state*)
	Error := TRUE;
	ErrorID := 16#05; (*Command aborted*)
END_IF

(*State machine*)
CASE uiFbState OF
	0:	;

	1:	IF (-3276.8 <=  TargetForce AND TargetForce <= 3276.7)
		THEN
			(*Streaming*)
			bTemp := Axis.PlcToDrv.MCHeader.0;
			Axis.PlcToDrv.MCHeader := uiCmdHeader;
			Axis.PlcToDrv.MCHeader.0 := NOT bTemp;
	
			(*Parameter Umrechung*)
			(*Calculate parameters*)
			Axis.PlcToDrv.MCParaWord0 := REAL_TO_UINT(TargetForce * 10); (*Target force*)
	
			Streaming := TRUE;

			IF NOT Enable THEN
				uiFbState := 3;
			END_IF
		ELSE
			Axis.CommandRunning := FALSE;
			uiFbState := 50; (*Error state*)
			Error := TRUE;
			ErrorID := 16#06; (*Invalid input(s)*)
		END_IF

	3:	IF Axis.PlcToDrv.MCHeader.0 = Axis.DrvToPlc.StateVar.0 THEN
			Streaming := FALSE;
			Axis.PlcToDrv.MCHeader := 16#0000; (*No Operation*)
			Axis.PlcToDrv.MCHeader.0 := Axis.DrvToPlc.StateVar.0;
			Axis.CommandRunning := FALSE;
		 	uiFbState := 0;
		END_IF

	50:	Error := TRUE;
		Axis.PlcToDrv.MCHeader := 16#0000; (*No Operation*)
		Streaming := FALSE;
		uiFbState := 51;

	51:	 IF NOT Enable THEN
			uiFbState := 0;
			Error := FALSE;
			ErrorID := 0;
		END_IF

END_CASE

END_FUNCTION_BLOCK

// POUs/LinMot Force Control Function Blocks/LMfc_ChangeTargetForce
FUNCTION_BLOCK LMfc_ChangeTargetForce
VAR_INPUT
	Execute			:BOOL;	(*Execute command*)
	TargetForce		:REAL;	(*Target force*)
END_VAR
VAR_IN_OUT
	Axis			:tstLM_Axis; (*Axis reference*)
END_VAR
VAR_OUTPUT
	Done			:BOOL;	(*Command has been executed*)
	Busy			:BOOL;	(*Command running / FB Busy*)
	Error			:BOOL;	(*Error detected*)
	ErrorID			:UINT;	(*Error ID:
							01h: Axis not ready
 							02h: Axis already has command running
 							03h: Axis has error
 							04h: Command interrupted
 							05h: Command aborted
							06h: Invalid input(s)
							*)
END_VAR
VAR
	usiOldCmdCount 	:USINT;	(*internal -> *)
	usiNewCmdCount	:USINT;	(*internal -> *)
	uiCState		:UINT;	(*internal -> *)
	uiFbState		:UINT;	(*internal -> *)
	rTrig			:LM_R_TRIG;	(*internal -> *)

 	uiCmdHeader 	:UINT := 16#3820;	(*CommandHeader (382xh) of the "Force Ctrl Change Target Force (382xh)" motion command*)
END_VAR
(*Version history:
Date         	 | Version    		| Created under     	| Author          	| Remark 
------------------------------------------------------------------------------------------------------------------------------- 
2011-sep-13   	 | 1.0.0      		| V2.11.0 (Build 1016)	| fj  				| initial release 
2011-dec-01   	 | 1.0.2      		| V2.11.0 (Build 1016)	| fj  				| code optimisation
2012-apr-25   	 | 1.1.0     		| V2.11.0 (Build 1016)	| fj  				| added input parameters check
*)

(*Variablen ][ variables*)
usiOldCmdCount := SHR(UINT_TO_USINT(SHL(Axis.DrvToPlc.StateVar,4)),4);
uiCState := SHR(Axis.DrvToPlc.StateVar, 8);

(*Flankenerkennung am Execute Eingang*)
(*Edge detection on Execute input*)
rTrig(CLK:=Execute);
IF rTrig.Q AND uiCState = 16#08 AND NOT Axis.CommandRunning THEN (*Start command*)
	Axis.CommandRunning := TRUE;
	Busy := TRUE;
	uiFbState := 1;
ELSIF rTrig.Q AND Busy THEN (*Restart command / New rising edge on execute input*)
	Axis.CommandRunning := TRUE;
	Busy := TRUE;
	uiFbState := 1;
ELSIF rTrig.Q AND uiCState <> 16#08 THEN (*Axis not ready*)
	uiFbState := 50; (*Error state*)
	Error := TRUE;
	ErrorID := 16#01; (*Axis not ready*)
ELSIF rTrig.Q AND Axis.CommandRunning AND NOT Busy THEN (*Axis already has a command running*)
	uiFbState := 50; (*Error state*)
	Error := TRUE;
	ErrorID := 16#02; (*Axis already has a command running*)
END_IF

IF Busy AND uiCState = 16#04 THEN
	Axis.CommandRunning := FALSE;
	uiFbState := 50;
	Error := TRUE;
	ErrorID := 16#03; (*Axis has error*)
END_IF

IF Busy AND uiCState <> 16#08 THEN
	Axis.CommandRunning := FALSE;
	uiFbState := 50; (*Error state*)
	Error := TRUE;
	ErrorID := 16#04; (*Command interupted*)
ELSIF Busy AND Axis.CommandAborted THEN
	uiFbState := 50; (*Error state*)
	Error := TRUE;
	ErrorID := 16#05; (*Command aborted*)
END_IF

(*State machine*)
CASE uiFbState OF
	0:	;

	1:	IF (-3276.8 <= TargetForce AND TargetForce <= 3276.7)
		THEN
			(*Befehlskopf mit CMD Count berechen und senden ][ Calculate and send command header*)
			usiNewCmdCount := (usiOldCmdCount + 1) MOD 16 ; (*MOD 16*)
			Axis.PlcToDrv.MCHeader := 16#0000; (*Reset Header*)
			Axis.PlcToDrv.MCHeader := uiCmdHeader + usiNewCmdCount;

			Axis.PlcToDrv.MCParaWord0 := REAL_TO_UINT(TargetForce * 10); (*Target force*)

			LM_UptMCI(Axis);

			uiFbState := 2;
		ELSE
			Axis.CommandRunning := FALSE;
			uiFbState := 50; (*Error state*)
			Error := TRUE;
			ErrorID := 16#06; (*Invalid input(s)*)
		END_IF

	2:	(*Prüfen ob Befehl ausgeführt ][ Check if command has been executed*)
		IF usiOldCmdCount = usiNewCmdCount AND uiCState = 16#08 THEN
			Done := TRUE;
			Busy := FALSE;
			Axis.PlcToDrv.MCHeader := 16#0000 + usiNewCmdCount; (*Send no operation*)
			Axis.CommandRunning := FALSE;
			uiFbState := 3;
		END_IF

	3:	IF NOT Execute THEN
			uiFbState := 0;
			Busy := FALSE;
			Done := FALSE;
		END_IF

	50:	Error := TRUE;
		Busy := FALSE;
		Done := FALSE;
		IF NOT Execute THEN
			uiFbState := 0;
			Error := FALSE;
			ErrorID := 0;
		END_IF

END_CASE

END_FUNCTION_BLOCK

// POUs/LinMot Force Control Function Blocks/LMfc_GoToPosForceCtrlHighLim
FUNCTION_BLOCK LMfc_GoToPosForceCtrlHighLim
VAR_INPUT
	Execute			:BOOL;	(*Execute command*)
	Position     	:REAL;	(*Target position in [mm]*)
	Velocity		:REAL;	(*Maximal velocity in [m/s]*)
	Acceleration   	:REAL;	(*Acceleration in [m/s^2]*)
	ForceLimit	   	:REAL;	(*Force limit [N]*)
	TargetForce	   	:REAL;	(*Target force [N]*)
END_VAR
VAR_IN_OUT
	Axis			:tstLM_Axis; (*Axis reference*)
END_VAR
VAR_OUTPUT
	Done			:BOOL;	(*Command has been executed*)
	Busy			:BOOL;	(*Command running / FB Busy*)
	Error			:BOOL;	(*Error detected*)
	ErrorID 		:UINT;	(*Error ID:
							01h: Axis not ready
 							02h: Axis already has command running
 							03h: Axis has error
 							04h: Command interrupted
 							05h: Command aborted
							06h: Invalid input(s)
							07h: Target Position reached but not switched to force control (Limit Force was not detected)
							*)
END_VAR
VAR
	usiOldCmdCount 	:USINT;	(*internal -> *)
	usiNewCmdCount	:USINT;	(*internal -> *)
	uiCState		:UINT;	(*internal -> *)
	uiFbState		:UINT;	(*internal -> *)
	rTrig			:LM_R_TRIG;	(*internal -> *)
	udiTmpDWord		:UDINT;	(*internal -> *)

 	uiCmdHeader 	:UINT := 16#3830;	(*CommandHeader (383xh) of the "VAI Go To Pos With Higher Force Ctrl Limit and Target Force (383xh)" motion command*)
END_VAR
(*Version history:
Date         	 | Version    		| Created under     	| Author          	| Remark 
------------------------------------------------------------------------------------------------------------------------------- 
2011-sep-13   	 | 1.0.0      		| V2.11.0 (Build 1016)	| fj  				| initial release 
2011-dec-01   	 | 1.0.2      		| V2.11.0 (Build 1016)	| fj  				| code optimisation
2012-oct-09   	 | 1.1.0     		| V2.11.0 (Build 1016)	| fj  				| added input parameters check, Done ouput is set if drive switches from position to force control. If not Error and ErrorID 16#07 is set
*)

(*Variablen ][ variables*)
usiOldCmdCount := SHR(UINT_TO_USINT(SHL(Axis.DrvToPlc.StateVar,4)),4);
uiCState := SHR(Axis.DrvToPlc.StateVar, 8);

(*Flankenerkennung am Execute Eingang*)
(*Edge detection on Execute input*)
rTrig(CLK:=Execute);
IF rTrig.Q AND uiCState = 16#08 AND NOT Axis.CommandRunning THEN (*Start command*)
	Axis.CommandRunning := TRUE;
	Busy := TRUE;
	uiFbState := 1;
ELSIF rTrig.Q AND Busy THEN (*Restart command / New rising edge on execute input*)
	Axis.CommandRunning := TRUE;
	Busy := TRUE;
	uiFbState := 1;
ELSIF rTrig.Q AND uiCState <> 16#08 THEN (*Axis not ready*)
	uiFbState := 50; (*Error state*)
	Error := TRUE;
	ErrorID := 16#01; (*Axis not ready*)
ELSIF rTrig.Q AND Axis.CommandRunning AND NOT Busy THEN (*Axis already has a command running*)
	uiFbState := 50; (*Error state*)
	Error := TRUE;
	ErrorID := 16#02; (*Axis already has a command running*)
END_IF

IF Busy AND uiCState = 16#04 THEN
	Axis.CommandRunning := FALSE;
	uiFbState := 50;
	Error := TRUE;
	ErrorID := 16#03; (*Axis has error*)
END_IF

IF Busy AND uiCState <> 16#08 THEN
	Axis.CommandRunning := FALSE;
	uiFbState := 50; (*Error state*)
	Error := TRUE;
	ErrorID := 16#04; (*Command interupted*)
ELSIF Busy AND Axis.CommandAborted THEN
	uiFbState := 50; (*Error state*)
	Error := TRUE;
	ErrorID := 16#05; (*Command aborted*)
END_IF

(*State machine*)
CASE uiFbState OF
	0:	;

	1:	(*Check inputs on valid value*)
		IF (-214748.0 <= Position AND Position <= 214748.0)
			AND (0 < Velocity AND Velocity <=2147)
			AND (0 < Acceleration AND Acceleration <= 21474)
			AND (-3276.8 <= ForceLimit AND ForceLimit <= 3276.7)
			AND (-3276.8 <= TargetForce AND TargetForce <= 3276.7)
			THEN
			(*Befehlskopf mit CMD Count berechen und senden ][ Calculate and send command header*)
			usiNewCmdCount := (usiOldCmdCount + 1) MOD 16 ; (*MOD 16*)
			Axis.PlcToDrv.MCHeader := 16#0000; (*Reset Header*)
			Axis.PlcToDrv.MCHeader := uiCmdHeader + usiNewCmdCount;

			udiTmpDWord := DINT_TO_UDINT(REAL_TO_DINT(Position * 10000)); (*Target position*)
			Axis.PlcToDrv.MCParaWord0 := UDINT_TO_UINT(udiTmpDWord);
			Axis.PlcToDrv.MCParaWord1 := UDINT_TO_UINT(ROR(udiTmpDWord,16));

			udiTmpDWord := DINT_TO_UDINT(REAL_TO_DINT(Velocity * 1000000)); (*Maximal velocity*)
			Axis.PlcToDrv.MCParaWord2 := UDINT_TO_UINT(udiTmpDWord);
			Axis.PlcToDrv.MCParaWord3 := UDINT_TO_UINT(ROR(udiTmpDWord,16));

			udiTmpDWord := DINT_TO_UDINT(REAL_TO_DINT(Acceleration * 100000)); (*Acceleration*)
			Axis.PlcToDrv.MCParaWord4 := UDINT_TO_UINT(udiTmpDWord);
			Axis.PlcToDrv.MCParaWord5 := UDINT_TO_UINT(ROR(udiTmpDWord,16));

			Axis.PlcToDrv.MCParaWord6 := REAL_TO_UINT(ForceLimit * 10); (*Force limit*)

			Axis.PlcToDrv.MCParaWord7 := REAL_TO_UINT(TargetForce * 10); (*Target force*)

			LM_UptMCI(Axis);

			uiFbState := 2;
		ELSE
			Axis.CommandRunning := FALSE;
			uiFbState := 50; (*Error state*)
			Error := TRUE;
			ErrorID := 16#06; (*Invalid input(s)*)
		END_IF

	2:	(*Prüfen ob Befehl ausgeführt ][ Check if command has been executed*)
		IF usiOldCmdCount = usiNewCmdCount AND uiCState = 16#08 AND NOT Axis.DrvToPlc.StatusWord.13 AND  Axis.DrvToPlc.StatusWord.9 THEN (*NOT MotionActive AND SpecialMotionActive set*)
			Done := TRUE;
			Busy := FALSE;
			Axis.PlcToDrv.MCHeader := 16#0000 + usiNewCmdCount; (*Send no operation*)
			Axis.CommandRunning := FALSE;
			uiFbState := 3;
		ELSIF usiOldCmdCount = usiNewCmdCount AND uiCState = 16#08 AND NOT Axis.DrvToPlc.StatusWord.13 AND  NOT Axis.DrvToPlc.StatusWord.9 THEN (*NOT MotionActive AND NOT SpecialMotionActive set*)
			Axis.CommandRunning := FALSE;
			uiFbState := 50; (*Error state*)
			Error := TRUE;
			ErrorID := 16#07; (*Target Position reached but not switched to force control (Limit Force was not detected)*)
		END_IF

	3:	IF NOT Execute THEN
			uiFbState := 0;
			Busy := FALSE;
			Done := FALSE;
		END_IF

	50:	Error := TRUE;
		Busy := FALSE;
		Done := FALSE;
		IF NOT Execute THEN
			uiFbState := 0;
			Error := FALSE;
			ErrorID := 0;
		END_IF

END_CASE

END_FUNCTION_BLOCK

// POUs/LinMot Force Control Function Blocks/LMfc_GoToPosForceCtrlLowLim
FUNCTION_BLOCK LMfc_GoToPosForceCtrlLowLim
VAR_INPUT
	Execute			:BOOL;	(*Execute command*)
	Position		:REAL;	(*Target position in [mm]*)
	Velocity		:REAL;	(*Maximal velocity in [m/s]*)
	Acceleration	:REAL;	(*Acceleration in [m/s^2]*)
	ForceLimit		:REAL;	(*Force limit [N]*)
	TargetForce		:REAL;	(*Target force [N]*)
END_VAR
VAR_IN_OUT
	Axis			:tstLM_Axis; (*Axis reference*)
END_VAR
VAR_OUTPUT
	Done			:BOOL;	(*Command has been executed*)
	Busy			:BOOL;	(*Command running / FB Busy*)
	Error			:BOOL;	(*Error detected*)
	ErrorID			:UINT;	(*Error ID:
							01h: Axis not ready
 							02h: Axis already has command running
 							03h: Axis has error
 							04h: Command interrupted
 							05h: Command aborted
							06h: Invalid input(s)
							07h: Target Position reached but not switched to force control (Limit Force was not detected)
							*)
END_VAR
VAR
	usiOldCmdCount 	:USINT;	(*internal -> *)
	usiNewCmdCount	:USINT;	(*internal -> *)
	uiCState		:UINT;	(*internal -> *)
	uiFbState		:UINT;	(*internal -> *)
	rTrig			:LM_R_TRIG;	(*internal -> *)
	udiTmpDWord		:UDINT;	(*internal -> *)

 	uiCmdHeader 	:UINT := 16#3850;	(*CommandHeader (385xh) of the "VAI Go To Pos With Lower Force Ctrl Limit and Target Force (385xh)" motion command*)
END_VAR
(*Version history:
Date         	 | Version    		| Created under     	| Author          	| Remark 
------------------------------------------------------------------------------------------------------------------------------- 
2011-sep-13   	 | 1.0.0      		| V2.11.0 (Build 1016)	| fj  				| initial release 
2011-dec-01   	 | 1.0.2      		| V2.11.0 (Build 1016)	| fj  				| code optimisation
2012-oct-09   	 | 1.1.0     		| V2.11.0 (Build 1016)	| fj  				| added input parameters check, Done ouput is set if drive switches from position to force control. If not Error and ErrorID 16#07 is set
*)

(*Variablen ][ variables*)
usiOldCmdCount := SHR(UINT_TO_USINT(SHL(Axis.DrvToPlc.StateVar,4)),4);
uiCState := SHR(Axis.DrvToPlc.StateVar, 8);

(*Flankenerkennung am Execute Eingang*)
(*Edge detection on Execute input*)
rTrig(CLK:=Execute);
IF rTrig.Q AND uiCState = 16#08 AND NOT Axis.CommandRunning THEN (*Start command*)
	Axis.CommandRunning := TRUE;
	Busy := TRUE;
	uiFbState := 1;
ELSIF rTrig.Q AND Busy THEN (*Restart command / New rising edge on execute input*)
	Axis.CommandRunning := TRUE;
	Busy := TRUE;
	uiFbState := 1;
ELSIF rTrig.Q AND uiCState <> 16#08 THEN (*Axis not ready*)
	uiFbState := 50; (*Error state*)
	Error := TRUE;
	ErrorID := 16#01; (*Axis not ready*)
ELSIF rTrig.Q AND Axis.CommandRunning AND NOT Busy THEN (*Axis already has a command running*)
	uiFbState := 50; (*Error state*)
	Error := TRUE;
	ErrorID := 16#02; (*Axis already has a command running*)
END_IF

IF Busy AND uiCState = 16#04 THEN
	Axis.CommandRunning := FALSE;
	uiFbState := 50;
	Error := TRUE;
	ErrorID := 16#03; (*Axis has error*)
END_IF

IF Busy AND uiCState <> 16#08 THEN
	Axis.CommandRunning := FALSE;
	uiFbState := 50; (*Error state*)
	Error := TRUE;
	ErrorID := 16#04; (*Command interupted*)
ELSIF Busy AND Axis.CommandAborted THEN
	uiFbState := 50; (*Error state*)
	Error := TRUE;
	ErrorID := 16#05; (*Command aborted*)
END_IF

(*State machine*)
CASE uiFbState OF
	0:	;

	1:	(*Check inputs on valid value*)
		IF (-214748.0 <= Position AND Position <= 214748.0)
			AND (0 < Velocity AND Velocity <=2147)
			AND (0 < Acceleration AND Acceleration <= 21474)
			AND (-3276.8 <= ForceLimit AND ForceLimit <= 3276.7)
			AND (-3276.8 <= TargetForce AND TargetForce <= 3276.7)
			THEN
			(*Befehlskopf mit CMD Count berechen und senden ][ Calculate and send command header*)
			usiNewCmdCount := (usiOldCmdCount + 1) MOD 16 ; (*MOD 16*)
			Axis.PlcToDrv.MCHeader := 16#0000; (*Reset Header*)
			Axis.PlcToDrv.MCHeader := uiCmdHeader + usiNewCmdCount;

			udiTmpDWord := DINT_TO_UDINT(REAL_TO_DINT(Position * 10000)); (*Target position*)
			Axis.PlcToDrv.MCParaWord0 := UDINT_TO_UINT(udiTmpDWord);
			Axis.PlcToDrv.MCParaWord1 := UDINT_TO_UINT(ROR(udiTmpDWord,16));

			udiTmpDWord := DINT_TO_UDINT(REAL_TO_DINT(Velocity * 1000000)); (*Maximal velocity*)
			Axis.PlcToDrv.MCParaWord2 := UDINT_TO_UINT(udiTmpDWord);
			Axis.PlcToDrv.MCParaWord3 := UDINT_TO_UINT(ROR(udiTmpDWord,16));

			udiTmpDWord := DINT_TO_UDINT(REAL_TO_DINT(Acceleration * 100000)); (*Acceleration*)
			Axis.PlcToDrv.MCParaWord4 := UDINT_TO_UINT(udiTmpDWord);
			Axis.PlcToDrv.MCParaWord5 := UDINT_TO_UINT(ROR(udiTmpDWord,16));

			Axis.PlcToDrv.MCParaWord6 := REAL_TO_UINT(ForceLimit * 10); (*Force limit*)

			Axis.PlcToDrv.MCParaWord7 := REAL_TO_UINT(TargetForce * 10); (*Target force*)

			LM_UptMCI(Axis);

			uiFbState := 2;
		ELSE
			Axis.CommandRunning := FALSE;
			uiFbState := 50; (*Error state*)
			Error := TRUE;
			ErrorID := 16#06; (*Invalid input(s)*)
		END_IF

	2:	(*Prüfen ob Befehl ausgeführt ][ Check if command has been executed*)
		IF usiOldCmdCount = usiNewCmdCount AND uiCState = 16#08 AND NOT Axis.DrvToPlc.StatusWord.13 AND  Axis.DrvToPlc.StatusWord.9 THEN (*NOT MotionActive AND SpecialMotionActive set*)
			Done := TRUE;
			Busy := FALSE;
			Axis.PlcToDrv.MCHeader := 16#0000 + usiNewCmdCount; (*Send no operation*)
			Axis.CommandRunning := FALSE;
			uiFbState := 3;
		ELSIF usiOldCmdCount = usiNewCmdCount AND uiCState = 16#08 AND NOT Axis.DrvToPlc.StatusWord.13 AND  NOT Axis.DrvToPlc.StatusWord.9 THEN (*NOT MotionActive AND NOT SpecialMotionActive set*)
			Axis.CommandRunning := FALSE;
			uiFbState := 50; (*Error state*)
			Error := TRUE;
			ErrorID := 16#07; (*Target Position reached but not switched to force control (Limit Force was not detected)*)
		END_IF

	3:	IF NOT Execute THEN
			uiFbState := 0;
			Busy := FALSE;
			Done := FALSE;
		END_IF

	50:	Error := TRUE;
		Busy := FALSE;
		Done := FALSE;
		IF NOT Execute THEN
			uiFbState := 0;
			Error := FALSE;
			ErrorID := 0;
		END_IF

END_CASE

END_FUNCTION_BLOCK

// POUs/LinMot Force Control Function Blocks/LMfc_GoToPosRstForceCtrl
FUNCTION_BLOCK LMfc_GoToPosRstForceCtrl
VAR_INPUT
	Execute			:BOOL;	(*Execute command*)
	Position		:REAL;	(*Target position in [mm]*)
	Velocity		:REAL;	(*Maximal velocity in [m/s]*)
	Acceleration	:REAL;	(*Acceleration in [m/s^2]*)
	Deceleration	:REAL;	(*Deceleration in [m/s^2]*)
END_VAR
VAR_IN_OUT
	Axis			:tstLM_Axis; (*Axis reference*)
END_VAR
VAR_OUTPUT
	Done			:BOOL;	(*Command has been executed*)
	Busy			:BOOL;	(*Command running / FB Busy*)
	Error			:BOOL;	(*Error detected*)
	ErrorID			:UINT;	(*Error ID:
							01h: Axis not ready
 							02h: Axis already has command running
 							03h: Axis has error
 							04h: Command interrupted
 							05h: Command aborted
							06h: Invalid input(s)
							*)
END_VAR
VAR
	usiOldCmdCount 	:USINT;	(*internal -> *)
	usiNewCmdCount	:USINT;	(*internal -> *)
	uiCState		:UINT;	(*internal -> *)
	uiFbState		:UINT;	(*internal -> *)
	rTrig			:LM_R_TRIG;	(*internal -> *)
	udiTmpDWord		:UDINT;	(*internal -> *)

 	uiCmdHeader 	:UINT := 16#3860;	(*CommandHeader (386xh) of the "VAI Go To Pos From Act Pos And Reset Force Control Set I (386xh)" motion command*)
END_VAR
(*Version history:
Date         	 | Version    		| Created under     	| Author          	| Remark 
------------------------------------------------------------------------------------------------------------------------------- 
2011-sep-13   	 | 1.0.0      		| V2.11.0 (Build 1016)	| fj  				| initial release 
2011-dec-01   	 | 1.0.2      		| V2.11.0 (Build 1016)	| fj  				| code optimisation
2012-apr-25   	 | 1.1.0     		| V2.11.0 (Build 1016)	| fj  				| added input parameters check
*)

(*Variablen ][ variables*)
usiOldCmdCount := SHR(UINT_TO_USINT(SHL(Axis.DrvToPlc.StateVar,4)),4);
uiCState := SHR(Axis.DrvToPlc.StateVar, 8);

(*Flankenerkennung am Execute Eingang*)
(*Edge detection on Execute input*)
rTrig(CLK:=Execute);
IF rTrig.Q AND uiCState = 16#08 AND NOT Axis.CommandRunning THEN (*Start command*)
	Axis.CommandRunning := TRUE;
	Busy := TRUE;
	uiFbState := 1;
ELSIF rTrig.Q AND Busy THEN (*Restart command / New rising edge on execute input*)
	Axis.CommandRunning := TRUE;
	Busy := TRUE;
	uiFbState := 1;
ELSIF rTrig.Q AND uiCState <> 16#08 THEN (*Axis not ready*)
	uiFbState := 50; (*Error state*)
	Error := TRUE;
	ErrorID := 16#01; (*Axis not ready*)
ELSIF rTrig.Q AND Axis.CommandRunning AND NOT Busy THEN (*Axis already has a command running*)
	uiFbState := 50; (*Error state*)
	Error := TRUE;
	ErrorID := 16#02; (*Axis already has a command running*)
END_IF

IF Busy AND uiCState = 16#04 THEN
	Axis.CommandRunning := FALSE;
	uiFbState := 50;
	Error := TRUE;
	ErrorID := 16#03; (*Axis has error*)
END_IF

IF Busy AND uiCState <> 16#08 THEN
	Axis.CommandRunning := FALSE;
	uiFbState := 50; (*Error state*)
	Error := TRUE;
	ErrorID := 16#04; (*Command interupted*)
ELSIF Busy AND Axis.CommandAborted THEN
	uiFbState := 50; (*Error state*)
	Error := TRUE;
	ErrorID := 16#05; (*Command aborted*)
END_IF

(*State machine*)
CASE uiFbState OF
	0:	;

	1:     	(*Check inputs on valid value*)
		IF (-214748.0 <= Position AND Position <= 214748.0)
			AND (0.0 < Velocity AND Velocity <=2147.0)
			AND (0.0 < Acceleration AND Acceleration <= 21474.0)
			AND (0.0 < Acceleration AND Acceleration <= 21474.0)
			THEN
			(*Befehlskopf mit CMD Count berechen und senden ][ Calculate and send command header*)
			usiNewCmdCount := (usiOldCmdCount + 1) MOD 16 ; (*MOD 16*)
			Axis.PlcToDrv.MCHeader := 16#0000; (*Reset Header*)
			Axis.PlcToDrv.MCHeader := uiCmdHeader + usiNewCmdCount;

			udiTmpDWord := DINT_TO_UDINT(REAL_TO_DINT(Position * 10000)); (*Target position*)
			Axis.PlcToDrv.MCParaWord0 := UDINT_TO_UINT(udiTmpDWord);
			Axis.PlcToDrv.MCParaWord1 := UDINT_TO_UINT(ROR(udiTmpDWord,16));

			udiTmpDWord := DINT_TO_UDINT(REAL_TO_DINT(Velocity * 1000000)); (*Maximal velocity*)
			Axis.PlcToDrv.MCParaWord2 := UDINT_TO_UINT(udiTmpDWord);
			Axis.PlcToDrv.MCParaWord3 := UDINT_TO_UINT(ROR(udiTmpDWord,16));

			udiTmpDWord := DINT_TO_UDINT(REAL_TO_DINT(Acceleration * 100000)); (*Acceleration*)
			Axis.PlcToDrv.MCParaWord4 := UDINT_TO_UINT(udiTmpDWord);
			Axis.PlcToDrv.MCParaWord5 := UDINT_TO_UINT(ROR(udiTmpDWord,16));

			udiTmpDWord := DINT_TO_UDINT(REAL_TO_DINT(Deceleration * 100000)); (*Deceleration*)
			Axis.PlcToDrv.MCParaWord6 := UDINT_TO_UINT(udiTmpDWord);
			Axis.PlcToDrv.MCParaWord7 := UDINT_TO_UINT(ROR(udiTmpDWord,16));

			LM_UptMCI(Axis);

			uiFbState := 2;
		ELSE
			Axis.CommandRunning := FALSE;
			uiFbState := 50; (*Error state*)
			Error := TRUE;
			ErrorID := 16#06; (*Invalid input(s)*)
		END_IF

	2:	(*Prüfen ob Befehl ausgeführt ][ Check if command has been executed*)
		IF usiOldCmdCount = usiNewCmdCount AND uiCState = 16#08 AND Axis.DrvToPlc.StateVar.6 THEN
			Done := TRUE;
			Busy := FALSE;
			Axis.PlcToDrv.MCHeader := 16#0000 + usiNewCmdCount; (*Send no operation*)
			Axis.CommandRunning := FALSE;
			uiFbState := 3;
		END_IF

	3:	IF NOT Execute THEN
			uiFbState := 0;
			Busy := FALSE;
			Done := FALSE;
		END_IF

	50:	Error := TRUE;
		Busy := FALSE;
		Done := FALSE;
		IF NOT Execute THEN
			uiFbState := 0;
			Error := FALSE;
			ErrorID := 0;
		END_IF

END_CASE

END_FUNCTION_BLOCK

// POUs/LinMot Functions/F_GetVersionLinMotLibrary
FUNCTION F_GetVersionLinMotLibrary : UINT
VAR_INPUT
       nVersionElement       :       INT;
END_VAR
VAR
END_VAR
(*Version history:
Date         	 | Version    		| Created under     	| Author          	| Remark 
------------------------------------------------------------------------------------------------------------------------------- 
2011-jul-12   	 | 1.0.0      		| V2.11.0 (Build 1016)	| fj  				| initial release 
2011-sep-13   	 | 1.0.1      		| V2.11.0 (Build 1016)	| fj  				| removed check in FBs for "StandStill_LM" on Execute or Enable rising edge
2011-dec-01   	 | 1.0.2      		| V2.11.0 (Build 1016)	| fj  				| code optimisation
2012-jan-25   	 | 1.0.3     		| V2.11.0 (Build 1016)	| fj  				| LMct_AxisCtrlE12x0 & LMct_AxisCtrl11x0: operation enabled output is now directly mapped to the status word bit 0
2012-oct-16  	 | 1.1.0      		| V2.11.0 (Build 1016)	| fj  				| - LMmt_Stop: If input Deleceration is <= 0 the deceleration is set to 10m/s^2 by default
																				| - Added input parameter check for function blocks
																				| - Added LMct_AxisControl (Replaces LMct_AxisCtrlE12x0 & LMct_AxisCtrl11x0 & LMct_AxisCtrlB1150ML)
																				| - LMct_AxisCtrlE12x0 & LMct_AxisCtrl11x0 & LMct_AxisCtrlB1150ML: Added additional StateVar check for 090Fh ("homing finished") when rehoming. Required for motors with absolute position sensors
																				| - unofficial -> official: CAM Function Blocks & Force Control Function Blocks
																				| - tstLM_Axis inlcudes now Warnword and DemandPosition of the drive
																				| Obsolete: LMct_AxisCtrlE12x0 & LMct_AxisCtrl11x0 & LMct_AxisCtrlB1150ML (Replaced by LMct_AxisControl), LMct_RdAxisCom & LMct_WrAxisCom, don't use in new applications. Drive inputs and outputs can be mapped directly to tstLM_Axis now!
2014-feb-03  	 | 1.1.1			| V2.11.0 (Build 1816)	| fj  				| - Added LM_F_Trig & LM_R_Trig as edge detection functions. All function blocks now use this trigger functions
																				| - LMcm_CAMCtrl: Fixed command done check for modes <> 2
																				| - LMmt_Stop: check "not motion active" instead of "in target position" -> press applications
																				| - Reorganized tstLM_DrvToPlc struct to be compatible with ARM based PLCs -> Requires re-mapping in the system manager
2014-may-13  	 | 1.0.0.1			| v3.1.4014.0			| fj  				| - Converted library to TC3
2014-oct-20  	 | 1.0.0.2			| v3.1.4014.0			| fj  				| - Added rotary motors function blocks
*)

CASE nVersionElement OF
	1: (*major number*)
       		F_GetVersionLinMotLibrary := 1;
	2: (*minor number*)
       		F_GetVersionLinMotLibrary := 0;
	3: (*revision number*)
      		F_GetVersionLinMotLibrary := 0;
	ELSE
   		F_GetVersionLinMotLibrary := 16#FFFF;
END_CASE

END_FUNCTION

// POUs/LinMot MC Function Blocks/LMmt_Stop
FUNCTION_BLOCK LMmt_Stop
VAR_INPUT
	Execute			:BOOL;	(*Execute command*)
	Deceleration	:REAL;	(*Stop deceleration in [m/s^2]*)
END_VAR
VAR_IN_OUT
	Axis			:tstLM_Axis; (*Axis reference*)
END_VAR
VAR_OUTPUT
	Done			:BOOL;	(*Command has been executed*)
	Busy			:BOOL;	(*Command running / FB Busy*)
	Error			:BOOL;	(*Error detected*)
	ErrorID			:UINT;	(*Error ID:
							01h: Axis not ready
 							02h: Axis already has command running
 							03h: Axis has error
 							04h: Command interrupted
 							05h: Command aborted
							06h: Invalid input(s)
							*)
END_VAR
VAR
	usiOldCmdCount 	:USINT;	(*internal -> *)
	usiNewCmdCount	:USINT;	(*internal -> *)
	uiCState		:UINT;	(*internal -> *)
	uiFbState		:UINT;	(*internal -> *)
	rTrig			:LM_R_TRIG;	(*internal -> *)
	udiTmpDWord		:UDINT;	(*internal -> *)
	rDeceleration	:REAL;	(*internal -> *)

 	uiCmdHeader 	:UINT := 16#0170;	(*CommandHeader (017xh) of the "VAI Stop (017xh)" motion command*)
END_VAR
(*Version history:
Date         	 | Version    		| Created under     	| Author          	| Remark 
------------------------------------------------------------------------------------------------------------------------------- 
2011-jul-12   	 | 1.0.0      		| V2.11.0 (Build 1016)	| fj  				| initial release 
2011-dec-01   	 | 1.0.2      		| V2.11.0 (Build 1016)	| fj  				| code optimisation
2012-apr-25   	 | 1.1.0     		| V2.11.0 (Build 1016)	| fj  				| added input parameters check: if input Deleceration is <= 0 or > 21474 the deceleration is set to 10m/s^2 by default
2013-jan-22   	 | 1.1.1     		| V2.11.0 (Build 1016)	| fj  				| check "not motion active" instead of "in target position" -> press applications
*)

(*Variablen ][ variables*)
usiOldCmdCount := SHR(UINT_TO_USINT(SHL(Axis.DrvToPlc.StateVar,4)),4);
uiCState := SHR(Axis.DrvToPlc.StateVar, 8);

(*Flankenerkennung am Execute Eingang*)
(*Edge detection on Execute input*)
rTrig(CLK:=Execute);
IF rTrig.Q AND uiCState = 16#08 THEN
	Axis.CommandRunning := TRUE;
	Axis.CommandAborted := TRUE;
	Axis.AxisState := Stopping_LM;
	Busy := TRUE;
	uiFbState := 1;
ELSIF rTrig.Q AND uiCState <> 16#08 THEN
	uiFbState := 50; (*Error state*)
	Error := TRUE;
	ErrorID := 16#01; (*Axis not ready*)
END_IF

IF Busy AND uiCState = 16#04 THEN
	Axis.CommandRunning := FALSE;
	uiFbState := 50;
	Error := TRUE;
	ErrorID := 16#03; (*Axis has error*)
END_IF

IF Busy AND uiCState <> 16#08 THEN
	Axis.CommandRunning := FALSE;
	uiFbState := 50; (*Error state*)
	Error := TRUE;
	ErrorID := 16#04; (*Command interupted*)
END_IF

(*State machine*)
CASE uiFbState OF
	0:	;

	1:	(*Befehlskopf mit CMD Count berechen und senden ][ Calculate and send command header*)
		usiNewCmdCount := (usiOldCmdCount + 1) MOD 16 ; (*MOD 16*)
		Axis.PlcToDrv.MCHeader := 16#0000; (*Reset Header*)
		Axis.PlcToDrv.MCHeader := uiCmdHeader + usiNewCmdCount;

		IF Deceleration <= 0.0 OR Deceleration > 21474 THEN
			rDeceleration := 10.0; (*In case of invalid input Deceleration value the stop deceleration is set to 10m/s^2 by default*)
		ELSE
			rDeceleration := Deceleration;
		END_IF

		udiTmpDWord := DINT_TO_UDINT(REAL_TO_DINT(rDeceleration * 100000)); (*Stop deceleration*)
		Axis.PlcToDrv.MCParaWord0 := UDINT_TO_UINT(udiTmpDWord);
		Axis.PlcToDrv.MCParaWord1 := UDINT_TO_UINT(ROR(udiTmpDWord,16));

		LM_UptMCI(Axis);

		uiFbState := 2;

	2:	(*Prüfen ob Befehl ausgeführt ][ Check if command has been executed*)
		IF usiOldCmdCount = usiNewCmdCount AND uiCState = 16#08 AND NOT Axis.DrvToPlc.StateVar.5 THEN
			Done := TRUE;
			Busy := FALSE;
			uiFbState := 3;
		END_IF

	3:	IF NOT Execute THEN
			uiFbState := 0;
			Busy := FALSE;
			Done := FALSE;
			Axis.PlcToDrv.MCHeader := 16#0000 + usiNewCmdCount; (*Send no operation*)
			Axis.AxisState := StandStill_LM;
			Axis.CommandAborted := FALSE;
			Axis.CommandRunning := FALSE;
		END_IF

	50:	Error := TRUE;
		Busy := FALSE;
		Done := FALSE;
		IF NOT Execute THEN
			uiFbState := 0;
			Error := FALSE;
			ErrorID := 0;
		END_IF

END_CASE

END_FUNCTION_BLOCK

// POUs/LinMot MC Function Blocks/Unofficial_Unsupported/LMmt_IncrTargetPos
FUNCTION_BLOCK LMmt_IncrTargetPos
VAR_INPUT
	Execute			:BOOL;	(*Execute command*)
	Distance		:REAL;	(*Position increment in [mm]*)
	Velocity		:REAL;	(*Maximal velocity in [m/s]*)
	Acceleration	:REAL;	(*Acceleration in [m/s^2]*)
	Deceleration	:REAL;	(*Deceleration in [m/s^2]*)
END_VAR
VAR_IN_OUT
	Axis			:tstLM_Axis; (*Axis reference*)
END_VAR
VAR_OUTPUT
	Done			:BOOL;	(*Command has been executed*)
	Busy			:BOOL;	(*Command running / FB Busy*)
	Error			:BOOL;	(*Error detected*)
	ErrorID			:UINT;	(*Error ID:
							01h: Axis not ready
 							02h: Axis already has command running
 							03h: Axis has error
 							04h: Command interrupted
 							05h: Command aborted
							06h: Invalid input(s)
							*)
END_VAR
VAR
	usiOldCmdCount 	:USINT;	(*internal -> *)
	usiNewCmdCount	:USINT;	(*internal -> *)
	uiCState		:UINT;	(*internal -> *)
	uiFbState		:UINT;	(*internal -> *)
	rTrig			:LM_R_TRIG;	(*internal -> *)
	udiTmpDWord		:UDINT;	(*internal -> *)

 	uiCmdHeader 	:UINT := 16#0120;	(*CommandHeader (012xh) of the "VAI Increment Target Pos (012xh)" motion command*)
END_VAR
(*Version history:
Date         	 | Version    		| Created under     	| Author          	| Remark 
------------------------------------------------------------------------------------------------------------------------------- 
2012-oct-16  	 | 1.1.0     		| V2.11.0 (Build 1016)	| fj  				| initial release
*)

(*Variablen ][ variables*)
usiOldCmdCount := SHR(UINT_TO_USINT(SHL(Axis.DrvToPlc.StateVar,4)),4);
uiCState := SHR(Axis.DrvToPlc.StateVar, 8);

(*Flankenerkennung am Execute Eingang*)
(*Edge detection on Execute input*)
rTrig(CLK:=Execute);
IF rTrig.Q AND uiCState = 16#08 AND NOT Axis.CommandRunning THEN (*Start command*)
	Axis.CommandRunning := TRUE;
	Busy := TRUE;
	uiFbState := 1;
ELSIF rTrig.Q AND Busy THEN (*Restart command / New rising edge on execute input*)
	Axis.CommandRunning := TRUE;
	Busy := TRUE;
	uiFbState := 1;
ELSIF rTrig.Q AND uiCState <> 16#08 THEN (*Axis not ready*)
	uiFbState := 50; (*Error state*)
	Error := TRUE;
	ErrorID := 16#01; (*Axis not ready*)
ELSIF rTrig.Q AND Axis.CommandRunning AND NOT Busy THEN (*Axis already has a command running*)
	uiFbState := 50; (*Error state*)
	Error := TRUE;
	ErrorID := 16#02; (*Axis already has a command running*)
END_IF

IF Busy AND uiCState = 16#04 THEN
	Axis.CommandRunning := FALSE;
	uiFbState := 50;
	Error := TRUE;
	ErrorID := 16#03; (*Axis has error*)
END_IF

IF Busy AND uiCState <> 16#08 THEN
	Axis.CommandRunning := FALSE;
	uiFbState := 50; (*Error state*)
	Error := TRUE;
	ErrorID := 16#04; (*Command interupted*)
ELSIF Busy AND Axis.CommandAborted THEN
	uiFbState := 50; (*Error state*)
	Error := TRUE;
	ErrorID := 16#05; (*Command aborted*)
END_IF

(*State machine*)
CASE uiFbState OF
	0:	;

	1:	(*Check inputs on valid value*)
		IF (-214748.0 <= Distance AND Distance <= 214748.0)
			AND (0.0 < Velocity AND Velocity <= 2147.0)
			AND (0.0 < Acceleration AND Acceleration <= 21474.0)
			AND (0.0 < Deceleration AND Deceleration <= 21474.0)
			THEN
			(*Befehlskopf mit CMD Count berechen und senden ][ Calculate and send command header*)
			usiNewCmdCount := (usiOldCmdCount + 1) MOD 16 ; (*MOD 16*)
			Axis.PlcToDrv.MCHeader := 16#0000; (*Reset Header*)
			Axis.PlcToDrv.MCHeader := uiCmdHeader + usiNewCmdCount;

			udiTmpDWord := DINT_TO_UDINT(REAL_TO_DINT(Distance * 10000)); (*Target position*)
			Axis.PlcToDrv.MCParaWord0 := UDINT_TO_UINT(udiTmpDWord);
			Axis.PlcToDrv.MCParaWord1 := UDINT_TO_UINT(ROR(udiTmpDWord,16));

			udiTmpDWord := DINT_TO_UDINT(REAL_TO_DINT(Velocity * 1000000)); (*Maximal velocity*)
			Axis.PlcToDrv.MCParaWord2 := UDINT_TO_UINT(udiTmpDWord);
			Axis.PlcToDrv.MCParaWord3 := UDINT_TO_UINT(ROR(udiTmpDWord,16));

			udiTmpDWord := DINT_TO_UDINT(REAL_TO_DINT(Acceleration * 100000)); (*Acceleration*)
			Axis.PlcToDrv.MCParaWord4 := UDINT_TO_UINT(udiTmpDWord);
			Axis.PlcToDrv.MCParaWord5 := UDINT_TO_UINT(ROR(udiTmpDWord,16));

			udiTmpDWord := DINT_TO_UDINT(REAL_TO_DINT(Deceleration * 100000)); (*Deceleration*)
			Axis.PlcToDrv.MCParaWord6 := UDINT_TO_UINT(udiTmpDWord);
			Axis.PlcToDrv.MCParaWord7 := UDINT_TO_UINT(ROR(udiTmpDWord,16));

			LM_UptMCI(Axis);

			uiFbState := 2;
		ELSE
			Axis.CommandRunning := FALSE;
			uiFbState := 50; (*Error state*)
			Error := TRUE;
			ErrorID := 16#06; (*Invalid input(s)*)
		END_IF

	2:	(*Prüfen ob Befehl ausgeführt ][ Check if command has been executed*)
		IF usiOldCmdCount = usiNewCmdCount AND uiCState = 16#08 AND Axis.DrvToPlc.StateVar.6 THEN
			Done := TRUE;
			Busy := FALSE;
			Axis.PlcToDrv.MCHeader := 16#0000 + usiNewCmdCount; (*Send no operation*)
			Axis.CommandRunning := FALSE;
			uiFbState := 3;
		END_IF

	3:	IF NOT Execute THEN
			uiFbState := 0;
			Busy := FALSE;
			Done := FALSE;
		END_IF

	50:	Error := TRUE;
		Busy := FALSE;
		Done := FALSE;
		IF NOT Execute THEN
			uiFbState := 0;
			Error := FALSE;
			ErrorID := 0;
		END_IF

END_CASE

END_FUNCTION_BLOCK

// POUs/LinMot MC Function Blocks/LMmt_GenericMC
FUNCTION_BLOCK LMmt_GenericMC
VAR_INPUT
	Execute			:BOOL;	(*Execute command*)
	MCHeader		:UINT;	(*Motion Command Header*)
	MCParaWord0		:UINT;	(*Motion Command Parameter Word 0*)
	MCParaWord1		:UINT;	(*Motion Command Parameter Word 1*)
	MCParaWord2		:UINT;	(*Motion Command Parameter Word 2*)
	MCParaWord3		:UINT;	(*Motion Command Parameter Word 3*)
	MCParaWord4		:UINT;	(*Motion Command Parameter Word 4*)
	MCParaWord5		:UINT;	(*Motion Command Parameter Word 5*)
	MCParaWord6		:UINT;	(*Motion Command Parameter Word 6*)
	MCParaWord7		:UINT;	(*Motion Command Parameter Word 7*)
	MCParaWord8		:UINT;	(*Motion Command Parameter Word 8*)
END_VAR
VAR_IN_OUT
	Axis			:tstLM_Axis; (*Axis reference*)
END_VAR
VAR_OUTPUT
	Done			:BOOL;	(*Command has been executed*)
	Busy			:BOOL;	(*Command running / FB Busy*)
	Error			:BOOL;	(*Error detected*)
	ErrorID			:UINT;	(*Error ID:
							01h: Axis not ready
 							02h: Axis already has command running
 							03h: Axis has error
 							04h: Command interrupted
 							05h: Command aborted
							06h: Invalid input(s)
							*)
END_VAR
VAR
	usiOldCmdCount 	:USINT;	(*internal -> *)
	usiNewCmdCount	:USINT;	(*internal -> *)
	uiCState		:UINT;	(*internal -> *)
	uiFbState		:UINT;	(*internal -> *)
	rTrig			:LM_R_TRIG;	(*internal -> *)
END_VAR
(*Version history:
Date         	 | Version    		| Created under     	| Author          	| Remark 
------------------------------------------------------------------------------------------------------------------------------- 
2011-jul-12   	 | 1.0.0      		| V2.11.0 (Build 1016)	| fj  				| initial release 
2011-sep-13   	 | 1.0.1      		| V2.11.0 (Build 1016)	| fj  				| removed check for "StandStill_LM" on Execute rising edge
2011-dec-01   	 | 1.0.2      		| V2.11.0 (Build 1016)	| fj  				| code optimisation
*)

(*Variablen ][ variables*)
usiOldCmdCount := SHR(UINT_TO_USINT(SHL(Axis.DrvToPlc.StateVar,4)),4);
uiCState := SHR(Axis.DrvToPlc.StateVar, 8);

(*Flankenerkennung am Execute Eingang*)
(*Edge detection on Execute input*)
rTrig(CLK:=Execute);
IF rTrig.Q AND uiCState = 16#08 AND NOT Axis.CommandRunning THEN (*Start command*)
	Axis.CommandRunning := TRUE;
	Busy := TRUE;
	uiFbState := 1;
ELSIF rTrig.Q AND Busy THEN (*Restart command / New rising edge on execute input*)
	Axis.CommandRunning := TRUE;
	Busy := TRUE;
	uiFbState := 1;
ELSIF rTrig.Q AND uiCState <> 16#08 THEN (*Axis not ready*)
	uiFbState := 50; (*Error state*)
	Error := TRUE;
	ErrorID := 16#01; (*Axis not ready*)
ELSIF rTrig.Q AND Axis.CommandRunning AND NOT Busy THEN (*Axis already has a command running*)
	uiFbState := 50; (*Error state*)
	Error := TRUE;
	ErrorID := 16#02; (*Axis already has a command running*)
END_IF

IF Busy AND uiCState = 16#04 THEN
	Axis.CommandRunning := FALSE;
	uiFbState := 50;
	Error := TRUE;
	ErrorID := 16#03; (*Axis has error*)
END_IF

IF Busy AND uiCState <> 16#08 THEN
	Axis.CommandRunning := FALSE;
	uiFbState := 50; (*Error state*)
	Error := TRUE;
	ErrorID := 16#04; (*Command interupted*)
ELSIF Busy AND Axis.CommandAborted THEN
	uiFbState := 50; (*Error state*)
	Error := TRUE;
	ErrorID := 16#05; (*Command aborted*)
END_IF

(*State machine*)
CASE uiFbState OF
	0:	;

	1:	(*Befehlskopf mit CMD Count berechen und senden ][ Calculate and send command header*)
		usiNewCmdCount := (usiOldCmdCount + 1) MOD 16 ; (*MOD 16*)
		Axis.PlcToDrv.MCHeader := 16#0000; (*Reset Header*)
		Axis.PlcToDrv.MCHeader := MCHeader + usiNewCmdCount ;

		Axis.PlcToDrv.MCParaWord0 := MCParaWord0;
		Axis.PlcToDrv.MCParaWord1 := MCParaWord1;

		Axis.PlcToDrv.MCParaWord2 := MCParaWord2;
		Axis.PlcToDrv.MCParaWord3 := MCParaWord3;

		Axis.PlcToDrv.MCParaWord4 := MCParaWord4;
		Axis.PlcToDrv.MCParaWord5 := MCParaWord5;

		Axis.PlcToDrv.MCParaWord6 := MCParaWord6;
		Axis.PlcToDrv.MCParaWord7 := MCParaWord7;

		Axis.PlcToDrv.MCParaWord8 := MCParaWord8;

		LM_UptMCI(Axis);

		uiFbState := 2;

	2:	(*Prüfen ob Befehl ausgeführt ][ Check if command has been executed*)
		IF usiOldCmdCount = usiNewCmdCount AND uiCState = 16#08 THEN
			Done := TRUE;
			Busy := FALSE;
			Axis.PlcToDrv.MCHeader := 16#0000 + usiNewCmdCount; (*Send no operation*)
			Axis.CommandRunning := FALSE;
			uiFbState := 3;
		END_IF

	3:	IF NOT Execute THEN
			uiFbState := 0;
			Busy := FALSE;
			Done := FALSE;
		END_IF

	50:	Error := TRUE;
		Busy := FALSE;
		Done := FALSE;
		IF NOT Execute THEN
			uiFbState := 0;
			Error := FALSE;
			ErrorID := 0;
		END_IF

END_CASE

END_FUNCTION_BLOCK

// POUs/LinMot MC Function Blocks/LMmt_IncrActPos
FUNCTION_BLOCK LMmt_IncrActPos
VAR_INPUT
	Execute			:BOOL;	(*Execute command*)
	Distance		:REAL;	(*Position increment in [mm]*)
	Velocity		:REAL;	(*Maximal velocity in [m/s]*)
	Acceleration	:REAL;	(*Acceleration in [m/s^2]*)
	Deceleration	:REAL;	(*Deceleration in [m/s^2]*)
END_VAR
VAR_IN_OUT
	Axis			:tstLM_Axis; (*Axis reference*)
END_VAR
VAR_OUTPUT
	Done			:BOOL;	(*Command has been executed*)
	Busy			:BOOL;	(*Command running / FB Busy*)
	Error			:BOOL;	(*Error detected*)
	ErrorID			:UINT;	(*Error ID:
							01h: Axis not ready
 							02h: Axis already has command running
 							03h: Axis has error
 							04h: Command interrupted
 							05h: Command aborted
							06h: Invalid input(s)
							*)
END_VAR
VAR
	usiOldCmdCount 	:USINT;	(*internal -> *)
	usiNewCmdCount	:USINT;	(*internal -> *)
	uiCState		:UINT;	(*internal -> *)
	uiFbState		:UINT;	(*internal -> *)
	rTrig			:LM_R_TRIG;	(*internal -> *)
	udiTmpDWord		:UDINT;	(*internal -> *)

 	uiCmdHeader 	:UINT := 16#0150;	(*CommandHeader (015xh) of the "VAI Increment Act Pos (015xh)" motion command*)
END_VAR
(*Version history:
Date         	 | Version    		| Created under     	| Author          	| Remark 
------------------------------------------------------------------------------------------------------------------------------- 
2012-oct-16  	 | 1.1.0     		| V2.11.0 (Build 1016)	| fj  				| initial release
*)

(*Variablen ][ variables*)
usiOldCmdCount := SHR(UINT_TO_USINT(SHL(Axis.DrvToPlc.StateVar,4)),4);
uiCState := SHR(Axis.DrvToPlc.StateVar, 8);

(*Flankenerkennung am Execute Eingang*)
(*Edge detection on Execute input*)
rTrig(CLK:=Execute);
IF rTrig.Q AND uiCState = 16#08 AND NOT Axis.CommandRunning THEN (*Start command*)
	Axis.CommandRunning := TRUE;
	Busy := TRUE;
	uiFbState := 1;
ELSIF rTrig.Q AND Busy THEN (*Restart command / New rising edge on execute input*)
	Axis.CommandRunning := TRUE;
	Busy := TRUE;
	uiFbState := 1;
ELSIF rTrig.Q AND uiCState <> 16#08 THEN (*Axis not ready*)
	uiFbState := 50; (*Error state*)
	Error := TRUE;
	ErrorID := 16#01; (*Axis not ready*)
ELSIF rTrig.Q AND Axis.CommandRunning AND NOT Busy THEN (*Axis already has a command running*)
	uiFbState := 50; (*Error state*)
	Error := TRUE;
	ErrorID := 16#02; (*Axis already has a command running*)
END_IF

IF Busy AND uiCState = 16#04 THEN
	Axis.CommandRunning := FALSE;
	uiFbState := 50;
	Error := TRUE;
	ErrorID := 16#03; (*Axis has error*)
END_IF

IF Busy AND uiCState <> 16#08 THEN
	Axis.CommandRunning := FALSE;
	uiFbState := 50; (*Error state*)
	Error := TRUE;
	ErrorID := 16#04; (*Command interupted*)
ELSIF Busy AND Axis.CommandAborted THEN
	uiFbState := 50; (*Error state*)
	Error := TRUE;
	ErrorID := 16#05; (*Command aborted*)
END_IF

(*State machine*)
CASE uiFbState OF
	0:	;

	1:	(*Check inputs on valid value*)
		IF (-214748.0 <= Distance AND Distance <= 214748.0)
			AND (0.0 < Velocity AND Velocity <= 2147.0)
			AND (0.0 < Acceleration AND Acceleration <= 21474.0)
			AND (0.0 < Deceleration AND Deceleration <= 21474.0)
			THEN
			(*Befehlskopf mit CMD Count berechen und senden ][ Calculate and send command header*)
			usiNewCmdCount := (usiOldCmdCount + 1) MOD 16 ; (*MOD 16*)
			Axis.PlcToDrv.MCHeader := 16#0000; (*Reset Header*)
			Axis.PlcToDrv.MCHeader := uiCmdHeader + usiNewCmdCount;

			udiTmpDWord := DINT_TO_UDINT(REAL_TO_DINT(Distance * 10000)); (*Target position*)
			Axis.PlcToDrv.MCParaWord0 := UDINT_TO_UINT(udiTmpDWord);
			Axis.PlcToDrv.MCParaWord1 := UDINT_TO_UINT(ROR(udiTmpDWord,16));

			udiTmpDWord := DINT_TO_UDINT(REAL_TO_DINT(Velocity * 1000000)); (*Maximal velocity*)
			Axis.PlcToDrv.MCParaWord2 := UDINT_TO_UINT(udiTmpDWord);
			Axis.PlcToDrv.MCParaWord3 := UDINT_TO_UINT(ROR(udiTmpDWord,16));

			udiTmpDWord := DINT_TO_UDINT(REAL_TO_DINT(Acceleration * 100000)); (*Acceleration*)
			Axis.PlcToDrv.MCParaWord4 := UDINT_TO_UINT(udiTmpDWord);
			Axis.PlcToDrv.MCParaWord5 := UDINT_TO_UINT(ROR(udiTmpDWord,16));

			udiTmpDWord := DINT_TO_UDINT(REAL_TO_DINT(Deceleration * 100000)); (*Deceleration*)
			Axis.PlcToDrv.MCParaWord6 := UDINT_TO_UINT(udiTmpDWord);
			Axis.PlcToDrv.MCParaWord7 := UDINT_TO_UINT(ROR(udiTmpDWord,16));

			LM_UptMCI(Axis);

			uiFbState := 2;
		ELSE
			Axis.CommandRunning := FALSE;
			uiFbState := 50; (*Error state*)
			Error := TRUE;
			ErrorID := 16#06; (*Invalid input(s)*)
		END_IF

	2:	(*Prüfen ob Befehl ausgeführt ][ Check if command has been executed*)
		IF usiOldCmdCount = usiNewCmdCount AND uiCState = 16#08 AND Axis.DrvToPlc.StateVar.6 THEN
			Done := TRUE;
			Busy := FALSE;
			Axis.PlcToDrv.MCHeader := 16#0000 + usiNewCmdCount; (*Send no operation*)
			Axis.CommandRunning := FALSE;
			uiFbState := 3;
		END_IF

	3:	IF NOT Execute THEN
			uiFbState := 0;
			Busy := FALSE;
			Done := FALSE;
		END_IF

	50:	Error := TRUE;
		Busy := FALSE;
		Done := FALSE;
		IF NOT Execute THEN
			uiFbState := 0;
			Error := FALSE;
			ErrorID := 0;
		END_IF

END_CASE

END_FUNCTION_BLOCK

// POUs/LinMot MC Function Blocks/LMmt_MoveAbs
FUNCTION_BLOCK LMmt_MoveAbs
VAR_INPUT
	Execute			:BOOL;	(*Execute command*)
	Position		:REAL;	(*Target position in [mm]*)
	Velocity		:REAL;	(*Maximal velocity in [m/s]*)
	Acceleration	:REAL;	(*Acceleration in [m/s^2]*)
	Deceleration	:REAL;	(*Deceleration in [m/s^2]*)
END_VAR
VAR_IN_OUT
	Axis			:tstLM_Axis; (*Axis reference*)
END_VAR
VAR_OUTPUT
	Done			:BOOL;	(*Command has been executed*)
	Busy			:BOOL;	(*Command running / FB Busy*)
	Error			:BOOL;	(*Error detected*)
	ErrorID			:UINT;	(*Error ID:
							01h: Axis not ready
 							02h: Axis already has command running
 							03h: Axis has error
 							04h: Command interrupted
 							05h: Command aborted
							06h: Invalid input(s)
							*)
END_VAR
VAR
	usiOldCmdCount 	:USINT;	(*internal -> *)
	usiNewCmdCount	:USINT;	(*internal -> *)
	uiCState		:UINT;	(*internal -> *)
	uiFbState		:UINT;	(*internal -> *)
	rTrig			:LM_R_TRIG;	(*internal -> *)
	udiTmpDWord		:UDINT;	(*internal -> *)

 	uiCmdHeader 	:UINT := 16#0100;	(*CommandHeader (010xh) of the "VAI Go To Position (010xh)" motion command*)
END_VAR
(*Version history:
Date         	 | Version    		| Created under     	| Author          	| Remark 
------------------------------------------------------------------------------------------------------------------------------- 
2011-jul-12   	 | 1.0.0      		| V2.11.0 (Build 1016)	| fj  				| initial release 
2011-sep-13   	 | 1.0.1      		| V2.11.0 (Build 1016)	| fj  				| removed check on "StandStill_LM"
2011-dec-01   	 | 1.0.2      		| V2.11.0 (Build 1016)	| fj  				| code optimisation
2012-apr-25   	 | 1.1.0     		| V2.11.0 (Build 1016)	| fj  				| added input parameters check
*)

(*Variablen ][ variables*)
usiOldCmdCount := SHR(UINT_TO_USINT(SHL(Axis.DrvToPlc.StateVar,4)),4);
uiCState := SHR(Axis.DrvToPlc.StateVar, 8);

(*Flankenerkennung am Execute Eingang*)
(*Edge detection on Execute input*)
rTrig(CLK:=Execute);
IF rTrig.Q AND uiCState = 16#08 AND NOT Axis.CommandRunning THEN (*Start command*)
	Axis.CommandRunning := TRUE;
	Busy := TRUE;
	uiFbState := 1;
ELSIF rTrig.Q AND Busy THEN (*Restart command / New rising edge on execute input*)
	Axis.CommandRunning := TRUE;
	Busy := TRUE;
	uiFbState := 1;
ELSIF rTrig.Q AND uiCState <> 16#08 THEN (*Axis not ready*)
	uiFbState := 50; (*Error state*)
	Error := TRUE;
	ErrorID := 16#01; (*Axis not ready*)
ELSIF rTrig.Q AND Axis.CommandRunning AND NOT Busy THEN (*Axis already has a command running*)
	uiFbState := 50; (*Error state*)
	Error := TRUE;
	ErrorID := 16#02; (*Axis already has a command running*)
END_IF

IF Busy AND uiCState = 16#04 THEN
	Axis.CommandRunning := FALSE;
	uiFbState := 50;
	Error := TRUE;
	ErrorID := 16#03; (*Axis has error*)
END_IF

IF Busy AND uiCState <> 16#08 THEN
	Axis.CommandRunning := FALSE;
	uiFbState := 50; (*Error state*)
	Error := TRUE;
	ErrorID := 16#04; (*Command interupted*)
ELSIF Busy AND Axis.CommandAborted THEN
	uiFbState := 50; (*Error state*)
	Error := TRUE;
	ErrorID := 16#05; (*Command aborted*)
END_IF

(*State machine*)
CASE uiFbState OF
	0:	;

	1:	(*Check inputs on valid value*)
		IF (-214748.0 <= Position AND Position <= 214748.0)
			AND (0.0 < Velocity AND Velocity <= 2147.0)
			AND (0.0 < Acceleration AND Acceleration <= 21474.0)
			AND (0.0 < Deceleration AND Deceleration <= 21474.0)
			THEN
			(*Befehlskopf mit CMD Count berechen und senden ][ Calculate and send command header*)
			usiNewCmdCount := (usiOldCmdCount + 1) MOD 16 ; (*MOD 16*)
			Axis.PlcToDrv.MCHeader := 16#0000; (*Reset Header*)
			Axis.PlcToDrv.MCHeader := uiCmdHeader + usiNewCmdCount;

			udiTmpDWord := DINT_TO_UDINT(REAL_TO_DINT(Position * 10000)); (*Target position*)
			Axis.PlcToDrv.MCParaWord0 := UDINT_TO_UINT(udiTmpDWord);
			Axis.PlcToDrv.MCParaWord1 := UDINT_TO_UINT(ROR(udiTmpDWord,16));

			udiTmpDWord := DINT_TO_UDINT(REAL_TO_DINT(Velocity * 1000000)); (*Maximal velocity*)
			Axis.PlcToDrv.MCParaWord2 := UDINT_TO_UINT(udiTmpDWord);
			Axis.PlcToDrv.MCParaWord3 := UDINT_TO_UINT(ROR(udiTmpDWord,16));

			udiTmpDWord := DINT_TO_UDINT(REAL_TO_DINT(Acceleration * 100000)); (*Acceleration*)
			Axis.PlcToDrv.MCParaWord4 := UDINT_TO_UINT(udiTmpDWord);
			Axis.PlcToDrv.MCParaWord5 := UDINT_TO_UINT(ROR(udiTmpDWord,16));

			udiTmpDWord := DINT_TO_UDINT(REAL_TO_DINT(Deceleration * 100000)); (*Deceleration*)
			Axis.PlcToDrv.MCParaWord6 := UDINT_TO_UINT(udiTmpDWord);
			Axis.PlcToDrv.MCParaWord7 := UDINT_TO_UINT(ROR(udiTmpDWord,16));

			LM_UptMCI(Axis);
			
			uiFbState := 2;
		ELSE
			Axis.CommandRunning := FALSE;
			uiFbState := 50; (*Error state*)
			Error := TRUE;
			ErrorID := 16#06; (*Invalid input(s)*)
		END_IF

	2:	(*Prüfen ob Befehl ausgeführt ][ Check if command has been executed*)
		IF usiOldCmdCount = usiNewCmdCount AND uiCState = 16#08 AND Axis.DrvToPlc.StateVar.6 THEN
			Done := TRUE;
			Busy := FALSE;
			Axis.PlcToDrv.MCHeader := 16#0000 + usiNewCmdCount; (*Send no operation*)
			Axis.CommandRunning := FALSE;
			uiFbState := 3;
		END_IF

	3:	IF NOT Execute THEN
			uiFbState := 0;
			Busy := FALSE;
			Done := FALSE;
		END_IF

	50:	Error := TRUE;
		Busy := FALSE;
		Done := FALSE;
		IF NOT Execute THEN
			uiFbState := 0;
			Error := FALSE;
			ErrorID := 0;
		END_IF

END_CASE

END_FUNCTION_BLOCK

// POUs/LinMot MC Function Blocks/LMmt_MoveRel
FUNCTION_BLOCK LMmt_MoveRel
VAR_INPUT
	Execute			:BOOL;	(*Execute command*)
	Distance		:REAL;	(*Position increment in [mm]*)
	Velocity		:REAL;	(*Maximal velocity in [m/s]*)
	Acceleration	:REAL;	(*Acceleration in [m/s^2]*)
	Deceleration	:REAL;	(*Deceleration in [m/s^2]*)
END_VAR
VAR_IN_OUT
	Axis			:tstLM_Axis; (*Axis reference*)
END_VAR
VAR_OUTPUT
	Done			:BOOL;	(*Command has been executed*)
	Busy			:BOOL;	(*Command running / FB Busy*)
	Error			:BOOL;	(*Error detected*)
	ErrorID			:UINT;	(*Error ID:
							01h: Axis not ready
 							02h: Axis already has command running
 							03h: Axis has error
 							04h: Command interrupted
 							05h: Command aborted
							06h: Invalid input(s)
							*)
END_VAR
VAR
	usiOldCmdCount 	:USINT;	(*internal -> *)
	usiNewCmdCount	:USINT;	(*internal -> *)
	uiCState		:UINT;	(*internal -> *)
	uiFbState		:UINT;	(*internal -> *)
	rTrig			:LM_R_TRIG;	(*internal -> *)
	udiTmpDWord		:UDINT;	(*internal -> *)

 	uiCmdHeader 	:UINT := 16#0110;	(*CommandHeader (011xh) of the "VAI Increment Dem Pos (011xh)" motion command*)
END_VAR
(*Version history:
Date         	 | Version    		| Created under     	| Author          	| Remark 
------------------------------------------------------------------------------------------------------------------------------- 
2011-jul-12   	 | 1.0.0      		| V2.11.0 (Build 1016)	| fj  				| initial release 
2011-sep-13   	 | 1.0.1      		| V2.11.0 (Build 1016)	| fj  				| removed check for "StandStill_LM" on Execute rising edge
2011-dec-01   	 | 1.0.2      		| V2.11.0 (Build 1016)	| fj  				| code optimisation
2012-apr-25   	 | 1.1.0     		| V2.11.0 (Build 1016)	| fj  				| added input parameters check
*)

(*Variablen ][ variables*)
usiOldCmdCount := SHR(UINT_TO_USINT(SHL(Axis.DrvToPlc.StateVar,4)),4);
uiCState := SHR(Axis.DrvToPlc.StateVar, 8);

(*Flankenerkennung am Execute Eingang*)
(*Edge detection on Execute input*)
rTrig(CLK:=Execute);
IF rTrig.Q AND uiCState = 16#08 AND NOT Axis.CommandRunning THEN (*Start command*)
	Axis.CommandRunning := TRUE;
	Busy := TRUE;
	uiFbState := 1;
ELSIF rTrig.Q AND Busy THEN (*Restart command / New rising edge on execute input*)
	Axis.CommandRunning := TRUE;
	Busy := TRUE;
	uiFbState := 1;
ELSIF rTrig.Q AND uiCState <> 16#08 THEN (*Axis not ready*)
	uiFbState := 50; (*Error state*)
	Error := TRUE;
	ErrorID := 16#01; (*Axis not ready*)
ELSIF rTrig.Q AND Axis.CommandRunning AND NOT Busy THEN (*Axis already has a command running*)
	uiFbState := 50; (*Error state*)
	Error := TRUE;
	ErrorID := 16#02; (*Axis already has a command running*)
END_IF

IF Busy AND uiCState = 16#04 THEN
	Axis.CommandRunning := FALSE;
	uiFbState := 50;
	Error := TRUE;
	ErrorID := 16#03; (*Axis has error*)
END_IF

IF Busy AND uiCState <> 16#08 THEN
	Axis.CommandRunning := FALSE;
	uiFbState := 50; (*Error state*)
	Error := TRUE;
	ErrorID := 16#04; (*Command interupted*)
ELSIF Busy AND Axis.CommandAborted THEN
	uiFbState := 50; (*Error state*)
	Error := TRUE;
	ErrorID := 16#05; (*Command aborted*)
END_IF

(*State machine*)
CASE uiFbState OF
	0:	;

	1:	(*Check inputs on valid value*)
		IF (-214748.0 <= Distance AND Distance <= 214748.0)
			AND (0.0 < Velocity AND Velocity <= 2147.0)
			AND (0.0 < Acceleration AND Acceleration <= 21474.0)
			AND (0.0 < Deceleration AND Deceleration <= 21474.0)
			THEN
			(*Befehlskopf mit CMD Count berechen und senden ][ Calculate and send command header*)
			usiNewCmdCount := (usiOldCmdCount + 1) MOD 16 ; (*MOD 16*)
			Axis.PlcToDrv.MCHeader := 16#0000; (*Reset Header*)
			Axis.PlcToDrv.MCHeader := uiCmdHeader + usiNewCmdCount;

			udiTmpDWord := DINT_TO_UDINT(REAL_TO_DINT(Distance * 10000)); (*Target position*)
			Axis.PlcToDrv.MCParaWord0 := UDINT_TO_UINT(udiTmpDWord);
			Axis.PlcToDrv.MCParaWord1 := UDINT_TO_UINT(ROR(udiTmpDWord,16));

			udiTmpDWord := DINT_TO_UDINT(REAL_TO_DINT(Velocity * 1000000)); (*Maximal velocity*)
			Axis.PlcToDrv.MCParaWord2 := UDINT_TO_UINT(udiTmpDWord);
			Axis.PlcToDrv.MCParaWord3 := UDINT_TO_UINT(ROR(udiTmpDWord,16));

			udiTmpDWord := DINT_TO_UDINT(REAL_TO_DINT(Acceleration * 100000)); (*Acceleration*)
			Axis.PlcToDrv.MCParaWord4 := UDINT_TO_UINT(udiTmpDWord);
			Axis.PlcToDrv.MCParaWord5 := UDINT_TO_UINT(ROR(udiTmpDWord,16));

			udiTmpDWord := DINT_TO_UDINT(REAL_TO_DINT(Deceleration * 100000)); (*Deceleration*)
			Axis.PlcToDrv.MCParaWord6 := UDINT_TO_UINT(udiTmpDWord);
			Axis.PlcToDrv.MCParaWord7 := UDINT_TO_UINT(ROR(udiTmpDWord,16));

			LM_UptMCI(Axis);

			uiFbState := 2;
		ELSE
			Axis.CommandRunning := FALSE;
			uiFbState := 50; (*Error state*)
			Error := TRUE;
			ErrorID := 16#06; (*Invalid input(s)*)
		END_IF

	2:	(*Prüfen ob Befehl ausgeführt ][ Check if command has been executed*)
		IF usiOldCmdCount = usiNewCmdCount AND uiCState = 16#08 AND Axis.DrvToPlc.StateVar.6 THEN
			Done := TRUE;
			Busy := FALSE;
			Axis.PlcToDrv.MCHeader := 16#0000 + usiNewCmdCount; (*Send no operation*)
			Axis.CommandRunning := FALSE;
			uiFbState := 3;
		END_IF

	3:	IF NOT Execute THEN
			uiFbState := 0;
			Busy := FALSE;
			Done := FALSE;
		END_IF

	50:	Error := TRUE;
		Busy := FALSE;
		Done := FALSE;
		IF NOT Execute THEN
			uiFbState := 0;
			Error := FALSE;
			ErrorID := 0;
		END_IF

END_CASE

END_FUNCTION_BLOCK

// POUs/LinMot MC Function Blocks/LMmt_StartCTCommand
FUNCTION_BLOCK LMmt_StartCTCommand
VAR_INPUT
	Execute			:BOOL;	(*Execute command*)
	CTEntryID		:UINT;	(*ID of the Command Table to be started*)
END_VAR
VAR_IN_OUT
	Axis			:tstLM_Axis; (*Axis reference*)
END_VAR
VAR_OUTPUT
	Done			:BOOL;	(*Command has been executed*)
	Busy			:BOOL;	(*Command running / FB Busy*)
	Error			:BOOL;	(*Error detected*)
	ErrorID			:UINT;	(*Error ID:
							01h: Axis not ready
 							02h: Axis already has command running
 							03h: Axis has error
 							04h: Command interrupted
 							05h: Command aborted
							06h: Invalid input(s)
							*)
END_VAR
VAR
	usiOldCmdCount 	:USINT;	(*internal -> *)
	usiNewCmdCount	:USINT;	(*internal -> *)
	uiCState		:UINT;	(*internal -> *)
	uiFbState		:UINT;	(*internal -> *)
	rTrig			:LM_R_TRIG;	(*internal -> *)

 	uiCmdHeader 	:UINT := 16#2000;	(*CommandHeader (200xh) of the "Start Command Table Command (200xh)" motion command*)
END_VAR
(*Version history:
Date         	 | Version    		| Created under     	| Author          	| Remark 
------------------------------------------------------------------------------------------------------------------------------- 
2011-jul-12   	 | 1.0.0      		| V2.11.0 (Build 1016)	| fj  				| initial release
2011-sep-13   	 | 1.0.1      		| V2.11.0 (Build 1016)	| fj  				| removed check for "StandStill_LM" on Execute rising edge 
2011-dec-01   	 | 1.0.2      		| V2.11.0 (Build 1016)	| fj  				| code optimisation
2012-apr-25   	 | 1.1.0     		| V2.11.0 (Build 1016)	| fj  				| added input parameters check
*)

(*Variablen ][ variables*)
usiOldCmdCount := SHR(UINT_TO_USINT(SHL(Axis.DrvToPlc.StateVar,4)),4);
uiCState := SHR(Axis.DrvToPlc.StateVar, 8);

(*Flankenerkennung am Execute Eingang*)
(*Edge detection on Execute input*)
rTrig(CLK:=Execute);
IF rTrig.Q AND uiCState = 16#08 AND NOT Axis.CommandRunning THEN (*Start command*)
	Axis.CommandRunning := TRUE;
	Busy := TRUE;
	uiFbState := 1;
ELSIF rTrig.Q AND Busy THEN (*Restart command / New rising edge on execute input*)
	Axis.CommandRunning := TRUE;
	Busy := TRUE;
	uiFbState := 1;
ELSIF rTrig.Q AND uiCState <> 16#08 THEN (*Axis not ready*)
	uiFbState := 50; (*Error state*)
	Error := TRUE;
	ErrorID := 16#01; (*Axis not ready*)
ELSIF rTrig.Q AND Axis.CommandRunning AND NOT Busy THEN (*Axis already has a command running*)
	uiFbState := 50; (*Error state*)
	Error := TRUE;
	ErrorID := 16#02; (*Axis already has a command running*)
END_IF

IF Busy AND uiCState = 16#04 THEN
	Axis.CommandRunning := FALSE;
	uiFbState := 50;
	Error := TRUE;
	ErrorID := 16#03; (*Axis has error*)
END_IF

IF Busy AND uiCState <> 16#08 THEN
	Axis.CommandRunning := FALSE;
	uiFbState := 50; (*Error state*)
	Error := TRUE;
	ErrorID := 16#04; (*Command interupted*)
ELSIF Busy AND Axis.CommandAborted THEN
	uiFbState := 50; (*Error state*)
	Error := TRUE;
	ErrorID := 16#05; (*Command aborted*)
END_IF

(*State machine*)
CASE uiFbState OF
	0:	;

	1:	(*Check inputs on valid value*)
		IF (1 <= CTEntryID AND CTEntryID <= 255)
			THEN
			(*Befehlskopf mit CMD Count berechen und senden ][ Calculate and send command header*)
			usiNewCmdCount := (usiOldCmdCount + 1) MOD 16 ; (*MOD 16*)
			Axis.PlcToDrv.MCHeader := 16#0000; (*Reset Header*)
			Axis.PlcToDrv.MCHeader := uiCmdHeader + usiNewCmdCount;

			Axis.PlcToDrv.MCParaWord0 := CTEntryID; (*CTEntryID (line number)*)

			LM_UptMCI(Axis);

			uiFbState := 2;
		ELSE
			Axis.CommandRunning := FALSE;
			uiFbState := 50; (*Error state*)
			Error := TRUE;
			ErrorID := 16#06; (*Invalid input(s)*)
		END_IF

	2:	(*Prüfen ob Befehl ausgeführt ][ Check if command has been executed*)
		IF usiOldCmdCount = usiNewCmdCount AND uiCState = 16#08 THEN
			Done := TRUE;
			Busy := FALSE;
			Axis.PlcToDrv.MCHeader := 16#0000 + usiNewCmdCount; (*Send no operation*)
			Axis.CommandRunning := FALSE;
			uiFbState := 3;
		END_IF

	3:	IF NOT Execute THEN
			uiFbState := 0;
			Busy := FALSE;
			Done := FALSE;
		END_IF

	50:	Error := TRUE;
		Busy := FALSE;
		Done := FALSE;
		IF NOT Execute THEN
			uiFbState := 0;
			Error := FALSE;
			ErrorID := 0;
		END_IF

END_CASE

END_FUNCTION_BLOCK

// POUs/LinMot MC Function Blocks/LMmt_WriteLivePar
FUNCTION_BLOCK LMmt_WriteLivePar
VAR_INPUT
	Execute			:BOOL;	(*Execute command*)
	UPID			:UINT;	(*Parameter ID (UPID = Unique Parameter ID*)
	UPIDValue		:DINT;	(*Parameter value*)
END_VAR
VAR_IN_OUT
	Axis			:tstLM_Axis; (*Axis reference*)
END_VAR
VAR_OUTPUT
	Done			:BOOL;	(*Command has been executed*)
	Busy			:BOOL;	(*Command running / FB Busy*)
	Error			:BOOL;	(*Error detected*)
	ErrorID			:UINT;	(*Error ID:
							01h: Axis not ready
 							02h: Axis already has command running
 							03h: Axis has error
 							04h: Command interrupted
 							05h: Command aborted
							06h: Invalid input(s)
							*)
END_VAR
VAR
	usiOldCmdCount 	:USINT;	(*internal -> *)
	usiNewCmdCount	:USINT;	(*internal -> *)
	uiCState		:UINT;	(*internal -> *)
	uiFbState		:UINT;	(*internal -> *)
	rTrig			:LM_R_TRIG;	(*internal -> *)
	udiTmpDWord		:UDINT;	(*internal -> *)

 	uiCmdHeader 	:UINT := 16#0020;	(*CommandHeader (002xh) of the "Write Live Parameter (002xh)" motion command*)
END_VAR
(*Version history:
Date         	 | Version    		| Created under     	| Author          	| Remark 
------------------------------------------------------------------------------------------------------------------------------- 
2011-jul-12   	 | 1.0.0      		| V2.11.0 (Build 1016)	| fj  				| initial release 
2011-dec-01   	 | 1.0.2      		| V2.11.0 (Build 1016)	| fj  				| code optimisation
2012-apr-25   	 | 1.1.0     		| V2.11.0 (Build 1016)	| fj  				| added input parameters check
*)

(*Variablen ][ variables*)
usiOldCmdCount := SHR(UINT_TO_USINT(SHL(Axis.DrvToPlc.StateVar,4)),4);
uiCState := SHR(Axis.DrvToPlc.StateVar, 8);

(*Flankenerkennung am Execute Eingang*)
(*Edge detection on Execute input*)
rTrig(CLK:=Execute);
IF rTrig.Q AND uiCState = 16#08 AND NOT Axis.CommandRunning THEN (*Start command*)
	Axis.CommandRunning := TRUE;
	Busy := TRUE;
	uiFbState := 1;
ELSIF rTrig.Q AND Busy THEN (*Restart command / New rising edge on execute input*)
	Axis.CommandRunning := TRUE;
	Busy := TRUE;
	uiFbState := 1;
ELSIF rTrig.Q AND uiCState <> 16#08 THEN (*Axis not ready*)
	uiFbState := 50; (*Error state*)
	Error := TRUE;
	ErrorID := 16#01; (*Axis not ready*)
ELSIF rTrig.Q AND Axis.CommandRunning AND NOT Busy THEN (*Axis already has a command running*)
	uiFbState := 50; (*Error state*)
	Error := TRUE;
	ErrorID := 16#02; (*Axis already has a command running*)
END_IF

IF Busy AND uiCState = 16#04 THEN
	Axis.CommandRunning := FALSE;
	uiFbState := 50;
	Error := TRUE;
	ErrorID := 16#03; (*Axis has error*)
END_IF

IF Busy AND uiCState <> 16#08 THEN
	Axis.CommandRunning := FALSE;
	uiFbState := 50; (*Error state*)
	Error := TRUE;
	ErrorID := 16#04; (*Command interupted*)
ELSIF Busy AND Axis.CommandAborted THEN
	uiFbState := 50; (*Error state*)
	Error := TRUE;
	ErrorID := 16#05; (*Command aborted*)
END_IF

(*State machine*)
CASE uiFbState OF
	0:	;

	1:	(*Check inputs on valid value*)
		IF (0 < UPID AND UPID <= 65535)
			AND (-2147483648 <= UPIDValue AND UPIDValue <= 2147483647)
			THEN
			(*Befehlskopf mit CMD Count berechen und senden ][ Calculate and send command header*)
			usiNewCmdCount  := (usiOldCmdCount + 1) MOD 16 ; (*MOD 16*)
			Axis.PlcToDrv.MCHeader := 16#0000; (*Reset Header*)
			Axis.PlcToDrv.MCHeader := uiCmdHeader + usiNewCmdCount;

			Axis.PlcToDrv.MCParaWord0 := UPID; (*UPID number*)

			udiTmpDWord := DINT_TO_UDINT(UPIDValue); (*UPID parameter value*)
			Axis.PlcToDrv.MCParaWord1 := UDINT_TO_UINT(udiTmpDWord);
			Axis.PlcToDrv.MCParaWord2 := UDINT_TO_UINT(ROR(udiTmpDWord,16));

			LM_UptMCI(Axis);

			uiFbState := 2;
		ELSE
			Axis.CommandRunning := FALSE;
			uiFbState := 50; (*Error state*)
			Error := TRUE;
			ErrorID := 16#06; (*Invalid input(s)*)
		END_IF

	2:	(*Prüfen ob Befehl ausgeführt ][ Check if command has been executed*)
		IF usiOldCmdCount = usiNewCmdCount AND uiCState = 16#08 THEN
			Done := TRUE;
			Busy := FALSE;
			Axis.PlcToDrv.MCHeader := 16#0000 + usiNewCmdCount; (*Send no operation*)
			Axis.CommandRunning := FALSE;
			uiFbState := 3;
		END_IF

	3:	IF NOT Execute THEN
			uiFbState := 0;
			Busy := FALSE;
			Done := FALSE;
		END_IF

	50:	Error := TRUE;
		Busy := FALSE;
		Done := FALSE;
		IF NOT Execute THEN
			uiFbState := 0;
			Error := FALSE;
			ErrorID := 0;
		END_IF

END_CASE

END_FUNCTION_BLOCK

// POUs/LinMot MC Function Blocks Advanced/Unofficial_Unsupported/LMav_PVStreamLREAL
FUNCTION_BLOCK LMav_PVStreamLREAL
VAR_INPUT
	Enable 			:BOOL;	(*Enable PV streaming*)
	Position		:LREAL;	(*Setpoint position in [mm]*)
	Velocity		:LREAL;	(*Setpoint velocity in [mm/s]*)
END_VAR
VAR_IN_OUT
	Axis 			:tstLM_Axis; (*Axis*)
END_VAR
VAR_OUTPUT
	Streaming 		:BOOL;	(*Streaming / FB Busy*)
	Error 			:BOOL;	(*Error detected*)
	ErrorID			:UINT;	(*Error ID:
							01h: Axis not ready
 							02h: Axis already has command running
 							03h: Axis has error
 							04h: Command interrupted
 							05h: Command aborted
							06h: Invalid input(s)
							*)
END_VAR
VAR
	uiCState		:UINT;	(*internal -> *)
	uiFbState 		:UINT;	(*internal -> *)
	rTrig 			:LM_R_TRIG;	(*internal -> *)
	udiTmpDWord		:UDINT;	(*internal -> *)
	bTemp			:BOOL;	(*internal -> *)

